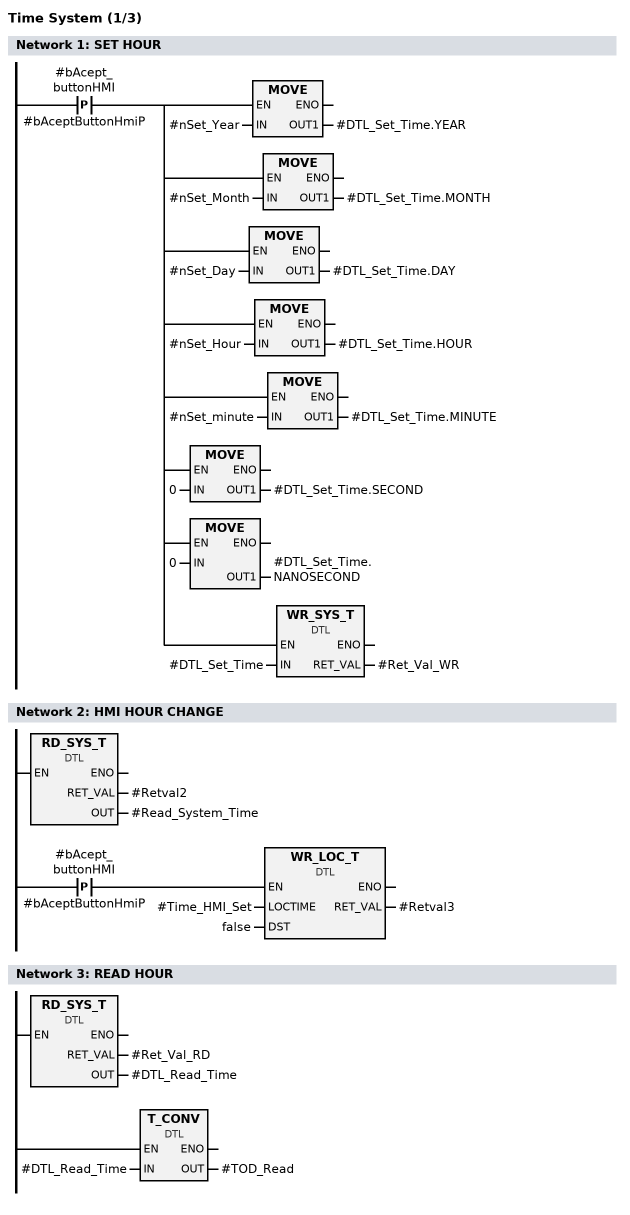
   RUNG wire#powerrail
      P_Contact(operand := #bAcept_buttonHMI, bit := #bAceptButtonHmiP)
      wire#w1
      Move(in := #nSet_Year, out1 => #DTL_Set_Time.YEAR)
   END_RUNG
   RUNG wire#w1
      Move(in := #nSet_Month, out1 => #DTL_Set_Time.MONTH)
   END_RUNG
   RUNG wire#w1
      Move(in := #nSet_Day, out1 => #DTL_Set_Time.DAY)
   END_RUNG
   RUNG wire#w1
      Move(in := #nSet_Hour, out1 => #DTL_Set_Time.HOUR)
   END_RUNG
   RUNG wire#w1
      Move(in := #nSet_minute, out1 => #DTL_Set_Time.MINUTE)
   END_RUNG
   RUNG wire#w1
      Move(in := 0, out1 => #DTL_Set_Time.SECOND)
   END_RUNG
   RUNG wire#w1
      Move(in := 0, out1 => #DTL_Set_Time.NANOSECOND)
   END_RUNG
   RUNG wire#w1
      { S7_Templates := "date_type := DTL" } WR_SYS_T(IN := #DTL_Set_Time, RET_VAL => #Ret_Val_WR)
   END_RUNG
   // the same network as SCL:
   #_w1 := #bAcept_buttonHMI AND NOT #bAceptButtonHmiP;   // rising edge of #bAcept_buttonHMI
   #bAceptButtonHmiP := #bAcept_buttonHMI;
   IF #_w1 THEN
       #DTL_Set_Time.YEAR := #nSet_Year;
       #DTL_Set_Time.MONTH := #nSet_Month;
       #DTL_Set_Time.DAY := #nSet_Day;
       #DTL_Set_Time.HOUR := #nSet_Hour;
       #DTL_Set_Time.MINUTE := #nSet_minute;
       #DTL_Set_Time.SECOND := 0;
       #DTL_Set_Time.NANOSECOND := 0;
       #Ret_Val_WR := WR_SYS_T(IN := #DTL_Set_Time);
   END_IF;
END_REGION

REGION Network 2: HMI HOUR CHANGE
   RUNG wire#powerrail
      { S7_Templates := "date_type := DTL" } RD_SYS_T(RET_VAL => #Retval2, OUT => #Read_System_Time)
   END_RUNG
   RUNG wire#powerrail
      P_Contact(operand := #bAcept_buttonHMI, bit := #bAceptButtonHmiP)
      { S7_Templates := "loctime_type := DTL" } WR_LOC_T(LOCTIME := #Time_HMI_Set, DST := false, Ret_Val => #Retval3)
   END_RUNG
   // the same network as SCL:
   #Retval2 := RD_SYS_T(OUT => #Read_System_Time);
   #_w1 := #bAcept_buttonHMI AND NOT #bAceptButtonHmiP;   // rising edge of #bAcept_buttonHMI
   #bAceptButtonHmiP := #bAcept_buttonHMI;
   IF #_w1 THEN #Retval3 := WR_LOC_T(LOCTIME := #Time_HMI_Set, DST := false); END_IF;
END_REGION

REGION Network 3: READ HOUR
   RUNG wire#powerrail
      { S7_Templates := "date_type := DTL" } RD_SYS_T(RET_VAL => #Ret_Val_RD, OUT => #DTL_Read_Time)
   END_RUNG
   RUNG wire#powerrail
      { S7_Templates := "[src_type := DTL, dest_type := Time_Of_Day]" } T_CONV(IN := #DTL_Read_Time, OUT => #TOD_Read)
   END_RUNG
   // the same network as SCL:
   #Ret_Val_RD := RD_SYS_T(OUT => #DTL_Read_Time);
   T_CONV(IN := #DTL_Read_Time, OUT => #TOD_Read);
END_REGION

REGION Network 4: WORK SHIFTS
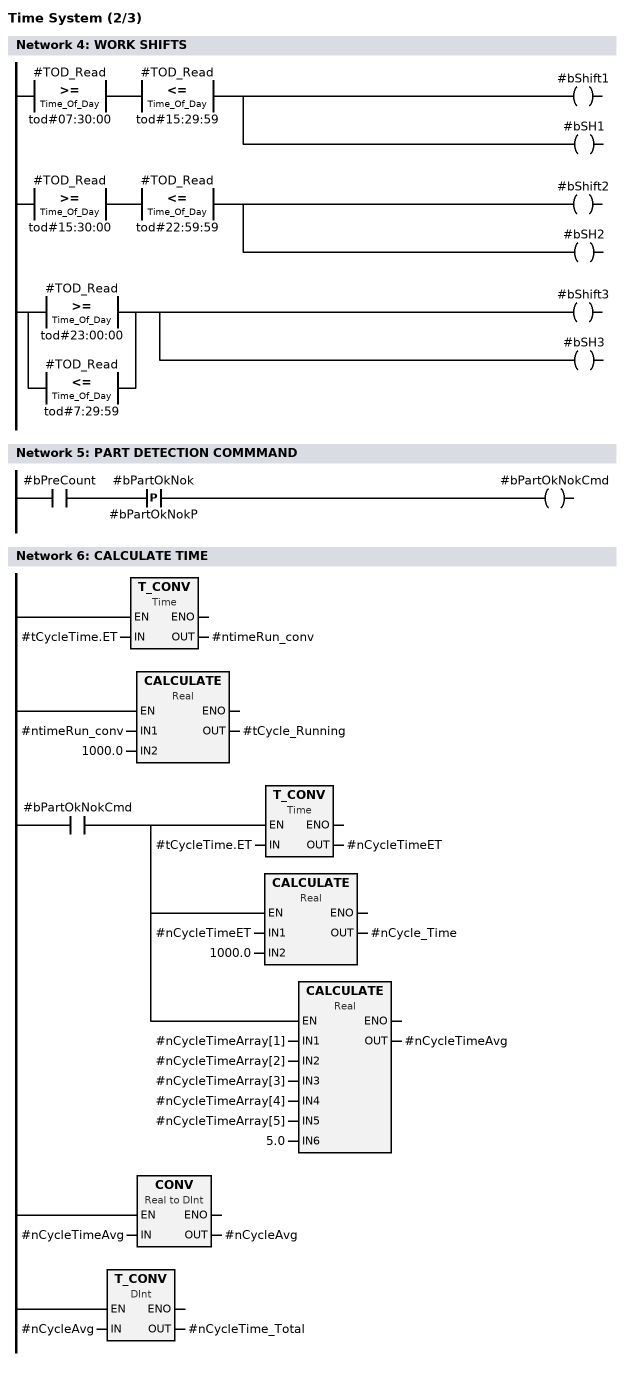
   RUNG wire#powerrail
      { S7_Templates := "SrcType := Time_Of_Day" } GE_Contact(in1 := #TOD_Read, in2 := tod#07:30:00)
      { S7_Templates := "SrcType := Time_Of_Day" } LE_Contact(in1 := #TOD_Read, in2 := tod#15:29:59)
      wire#w1
      Coil( #bShift1 )
   END_RUNG
   RUNG wire#w1
      Coil( #bSH1 )
   END_RUNG
   RUNG wire#powerrail
      { S7_Templates := "SrcType := Time_Of_Day" } GE_Contact(in1 := #TOD_Read, in2 := tod#15:30:00)
      { S7_Templates := "SrcType := Time_Of_Day" } LE_Contact(in1 := #TOD_Read, in2 := tod#22:59:59)
      wire#w2
      Coil( #bShift2 )
   END_RUNG
   RUNG wire#w2
      Coil( #bSH2 )
   END_RUNG
   RUNG wire#powerrail
      { S7_Templates := "SrcType := Time_Of_Day" } GE_Contact(in1 := #TOD_Read, in2 := tod#23:00:00)
      wire#w3
      Coil( #bShift3 )
   END_RUNG
   RUNG wire#powerrail
      { S7_Templates := "SrcType := Time_Of_Day" } LE_Contact(in1 := #TOD_Read, in2 := tod#7:29:59)
   END_RUNG wire#w3
   RUNG wire#w3
      Coil( #bSH3 )
   END_RUNG
   // the same network as SCL:
   #bShift1 := (#TOD_Read >= tod#07:30:00) AND (#TOD_Read <= tod#15:29:59);
   #bSH1 := #bShift1;
   #bShift2 := (#TOD_Read >= tod#15:30:00) AND (#TOD_Read <= tod#22:59:59);
   #bSH2 := #bShift2;
   #bShift3 := (#TOD_Read >= tod#23:00:00) OR (#TOD_Read <= tod#7:29:59);
   #bSH3 := #bShift3;
END_REGION

REGION Network 5: PART DETECTION COMMMAND
   RUNG wire#powerrail
      Contact( #bPreCount )
      P_Contact(operand := #bPartOkNok, bit := #bPartOkNokP)
      Coil( #bPartOkNokCmd )
   END_RUNG
   // the same network as SCL:
   #_w1 := #bPreCount AND #bPartOkNok AND NOT #bPartOkNokP;   // rising edge of #bPartOkNok
   #bPartOkNokP := #bPartOkNok;
   #bPartOkNokCmd := #_w1;
END_REGION

REGION Network 6: CALCULATE TIME
   RUNG wire#powerrail
      { S7_Templates := "[src_type := Time, dest_type := UDInt]" } T_CONV(IN := #tCycleTime.ET, OUT => #ntimeRun_conv)
   END_RUNG
   RUNG wire#powerrail
      { S7_Templates := "SrcType := Real"; S7_Expression := "in1/in2" } Calculate(in1 := #ntimeRun_conv, in2 := 1000.0, out => #tCycle_Running)
   END_RUNG
   RUNG wire#powerrail
      Contact( #bPartOkNokCmd )
      wire#w1
      { S7_Templates := "[src_type := Time, dest_type := UDInt]" } T_CONV(IN := #tCycleTime.ET, OUT => #nCycleTimeET)
   END_RUNG
   RUNG wire#w1
      { S7_Templates := "SrcType := Real"; S7_Expression := "in1/in2" } Calculate(in1 := #nCycleTimeET, in2 := 1000.0, out => #nCycle_Time)
   END_RUNG
   RUNG wire#w1
      { S7_Templates := "SrcType := Real"; S7_Expression := "(in1+in2+in3+in4+in5)/in6" } Calculate(in1 := #nCycleTimeArray[1], in2 := #nCycleTimeArray[2], in3 := #nCycleTimeArray[3], in4 := #nCycleTimeArray[4], in5 := #nCycleTimeArray[5], in6 := 5.0, out => #nCycleTimeAvg)
   END_RUNG
   RUNG wire#powerrail
      { S7_Templates := "[SrcType := Real, DestType := DInt]" } Convert(in := #nCycleTimeAvg, out => #nCycleAvg)
   END_RUNG
   RUNG wire#powerrail
      { S7_Templates := "[src_type := DInt, dest_type := Time_Of_Day]" } T_CONV(IN := #nCycleAvg, OUT => #nCycleTime_Total)
   END_RUNG
   // the same network as SCL:
   T_CONV(IN := #tCycleTime.ET, OUT => #ntimeRun_conv);
   #tCycle_Running := #ntimeRun_conv/1000.0;
   IF #bPartOkNokCmd THEN
       T_CONV(IN := #tCycleTime.ET, OUT => #nCycleTimeET);
       #nCycle_Time := #nCycleTimeET/1000.0;
       #nCycleTimeAvg := (#nCycleTimeArray[1]+#nCycleTimeArray[2]+#nCycleTimeArray[3]+#nCycleTimeArray[4]+#nCycleTimeArray[5])/5.0;
   END_IF;
   #nCycleAvg := REAL_TO_DINT(#nCycleTimeAvg);
   T_CONV(IN := #nCycleAvg, OUT => #nCycleTime_Total);
END_REGION

REGION Network 7: CICLE TIME ARRANGEMENT
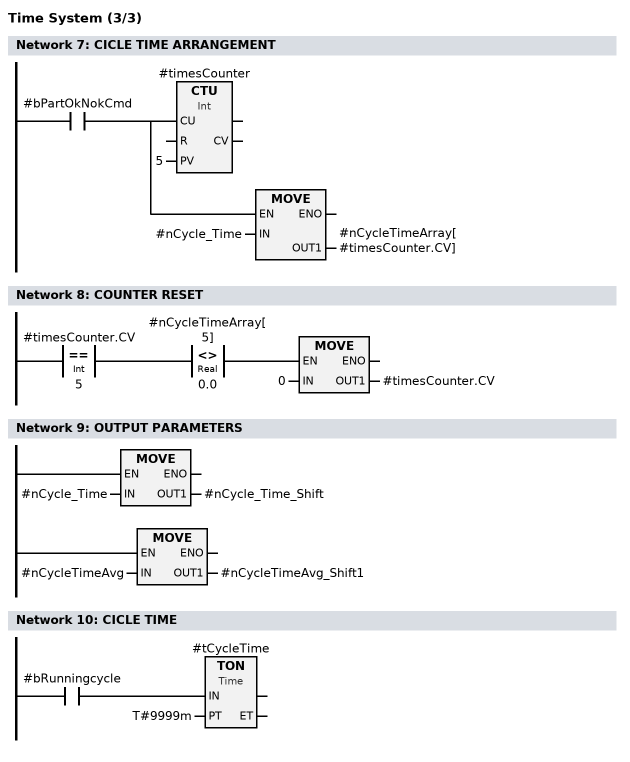
   RUNG wire#powerrail
      Contact( #bPartOkNokCmd )
      wire#w1
      { S7_Templates := "value_type := Int" } #timesCounter.CTU(r :=, pv := 5, cv =>)
   END_RUNG
   RUNG wire#w1
      Move(in := #nCycle_Time, out1 => #nCycleTimeArray[#timesCounter.CV])
   END_RUNG
   // the same network as SCL:
   #timesCounter.CTU(CU := #bPartOkNokCmd, PV := 5);
   IF #bPartOkNokCmd THEN #nCycleTimeArray[#timesCounter.CV] := #nCycle_Time; END_IF;
END_REGION

REGION Network 8: COUNTER RESET
   RUNG wire#powerrail
      { S7_Templates := "SrcType := Int" } EQ_Contact(in1 := #timesCounter.CV, in2 := 5)
      { S7_Templates := "SrcType := Real" } NE_Contact(in1 := #nCycleTimeArray[5], in2 := 0.0)
      Move(in := 0, out1 => #timesCounter.CV)
   END_RUNG
   // the same network as SCL:
   IF (#timesCounter.CV = 5) AND (#nCycleTimeArray[5] <> 0.0) THEN #timesCounter.CV := 0; END_IF;
END_REGION

REGION Network 9: OUTPUT PARAMETERS
   RUNG wire#powerrail
      Move(in := #nCycle_Time, out1 => #nCycle_Time_Shift)
   END_RUNG
   RUNG wire#powerrail
      Move(in := #nCycleTimeAvg, out1 => #nCycleTimeAvg_Shift1)
   END_RUNG
   // the same network as SCL:
   #nCycle_Time_Shift := #nCycle_Time;
   #nCycleTimeAvg_Shift1 := #nCycleTimeAvg;
END_REGION

REGION Network 10: CICLE TIME
   RUNG wire#powerrail
      Contact( #bRunningcycle )
      { S7_Templates := "time_type := Time" } #tCycleTime.TON(pt := T#9999m, et =>)
   END_RUNG
   // the same network as SCL:
   #tCycleTime.TON(IN := #bRunningcycle, PT := T#9999m);
END_REGION
END_FUNCTION_BLOCK

FUNCTION "FC_EKS" : Void   // FC305, LAD
TITLE = Euchner Management EKS KEY
{ S7_Optimized_Access := 'FALSE' }
VERSION : 0.1
// stored: AutoNumber false, IsIECCheckEnabled false, SetENOAutomatically false, UDAEnableTagReadback false
   VAR_INPUT
      iKEY_IN : Bool;
      iEKS_LEVEL : Byte;
      iEKS_EMPLOYEE_ID : DWord;
      iEKS_KEY_ID1 : DWord;
      iEKS_KEY_ID2 : DWord;
      iEKS_JOB_FINISHED : Bool;
      "Current_page_of HMI" : Word;
   END_VAR
   VAR_OUTPUT
      qEKS_START_ADDRESS : Byte;
      qEKS_DATA_LENGTH : Byte;
      qEKS_DATA_1 : Byte;
      qEKS_DATA_2 : DWord;
      qEKS_WRITE_CMD : Bool;
   END_VAR
   VAR_TEMP
      tNone : Bool;
      tDBAddressKeys : Int;
      tDBAddressHMIPage : Int;
      tDBKeyStructLength : Int;
      tDBAddress : Int;
      tDBLength : Int;
      tCycle : Int;
      tFill : Int;
      tKey : "udt_EKS_KEY";
      tDBStartAddress : Int;
      tsearch : Bool;
      i : Int;
   END_VAR
   VAR CONSTANT
      DB : Byte := 16#84;
   END_VAR
   VAR_TEMP   // added for the SCL form of the ladder/FBD networks
      _w1 : Bool;
      _w2 : Bool;
   END_VAR
BEGIN

REGION Network 1: Actual HMI page index limits
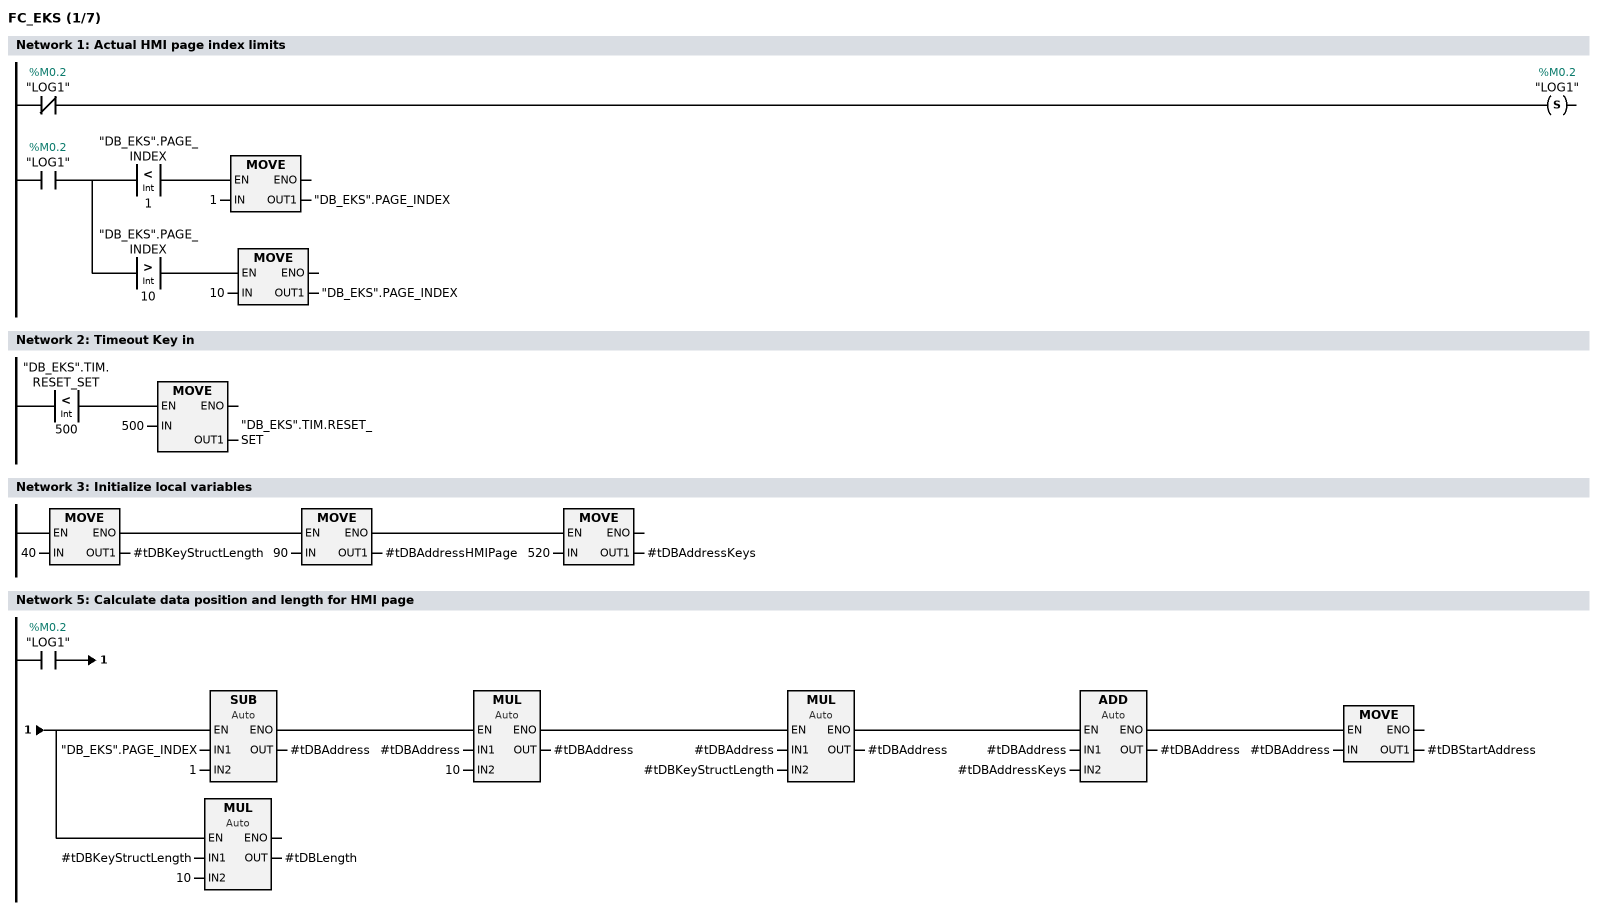
   RUNG wire#powerrail
      I_Contact( "LOG1" )
      S_Coil( "LOG1" )
   END_RUNG
   RUNG wire#powerrail
      Contact( "LOG1" )
      wire#w1
      { S7_Templates := "SrcType := Int" } LT_Contact(in1 := "DB_EKS".PAGE_INDEX, in2 := 1)
      Move(in := 1, out1 => "DB_EKS".PAGE_INDEX)
   END_RUNG
   RUNG wire#w1
      { S7_Templates := "SrcType := Int" } GT_Contact(in1 := "DB_EKS".PAGE_INDEX, in2 := 10)
      Move(in := 10, out1 => "DB_EKS".PAGE_INDEX)
   END_RUNG
   // the same network as SCL:
   IF NOT "LOG1" THEN "LOG1" := TRUE; END_IF;
   IF "LOG1" AND ("DB_EKS".PAGE_INDEX < 1) THEN "DB_EKS".PAGE_INDEX := 1; END_IF;
   IF "LOG1" AND ("DB_EKS".PAGE_INDEX > 10) THEN "DB_EKS".PAGE_INDEX := 10; END_IF;
END_REGION

REGION Network 2: Timeout Key in
   RUNG wire#powerrail
      { S7_Templates := "SrcType := Int" } LT_Contact(in1 := "DB_EKS".TIM.RESET_SET, in2 := 500)
      Move(in := 500, out1 => "DB_EKS".TIM.RESET_SET)
   END_RUNG
   // the same network as SCL:
   IF "DB_EKS".TIM.RESET_SET < 500 THEN "DB_EKS".TIM.RESET_SET := 500; END_IF;
END_REGION

REGION Network 3: Initialize local variables
   RUNG wire#powerrail
      Move(in := 40, out1 => #tDBKeyStructLength)
      Move(in := 90, out1 => #tDBAddressHMIPage)
      Move(in := 520, out1 => #tDBAddressKeys)
   END_RUNG
   // the same network as SCL:
   #tDBKeyStructLength := 40;
   #tDBAddressHMIPage := 90;
   #tDBAddressKeys := 520;
END_REGION

REGION Network 5: Calculate data position and length for HMI page
   RUNG wire#powerrail
      Contact( "LOG1" )
      wire#w1
      Sub(in1 := "DB_EKS".PAGE_INDEX, in2 := 1, out => #tDBAddress)
      Mul(in1 := #tDBAddress, in2 := 10, out => #tDBAddress)
      Mul(in1 := #tDBAddress, in2 := #tDBKeyStructLength, out => #tDBAddress)
      Add(in1 := #tDBAddress, in2 := #tDBAddressKeys, out => #tDBAddress)
      Move(in := #tDBAddress, out1 => #tDBStartAddress)
   END_RUNG
   RUNG wire#w1
      Mul(in1 := #tDBKeyStructLength, in2 := 10, out => #tDBLength)
   END_RUNG
   // the same network as SCL:
   IF "LOG1" THEN
       #tDBAddress := "DB_EKS".PAGE_INDEX - 1;
       #tDBAddress := #tDBAddress * 10;
       #tDBAddress := #tDBAddress * #tDBKeyStructLength;
       #tDBAddress := #tDBAddress + #tDBAddressKeys;
       #tDBStartAddress := #tDBAddress;
       #tDBLength := #tDBKeyStructLength * 10;
   END_IF;
END_REGION

REGION Network 6 (SCL): Copy data for page (10 keys)
   POKE_BLK(area_src:=#DB,
            dbNumber_src:=305,
            byteOffset_src:=#tDBAddress,
            area_dest:=#DB,
            dbNumber_dest:=305,
            byteOffset_dest:=90,
            count:=#tDBLength);
END_REGION

REGION Network 8: Inserted key
   // Store_Key_In is used to display only 1 time the level of euchner during storage function.
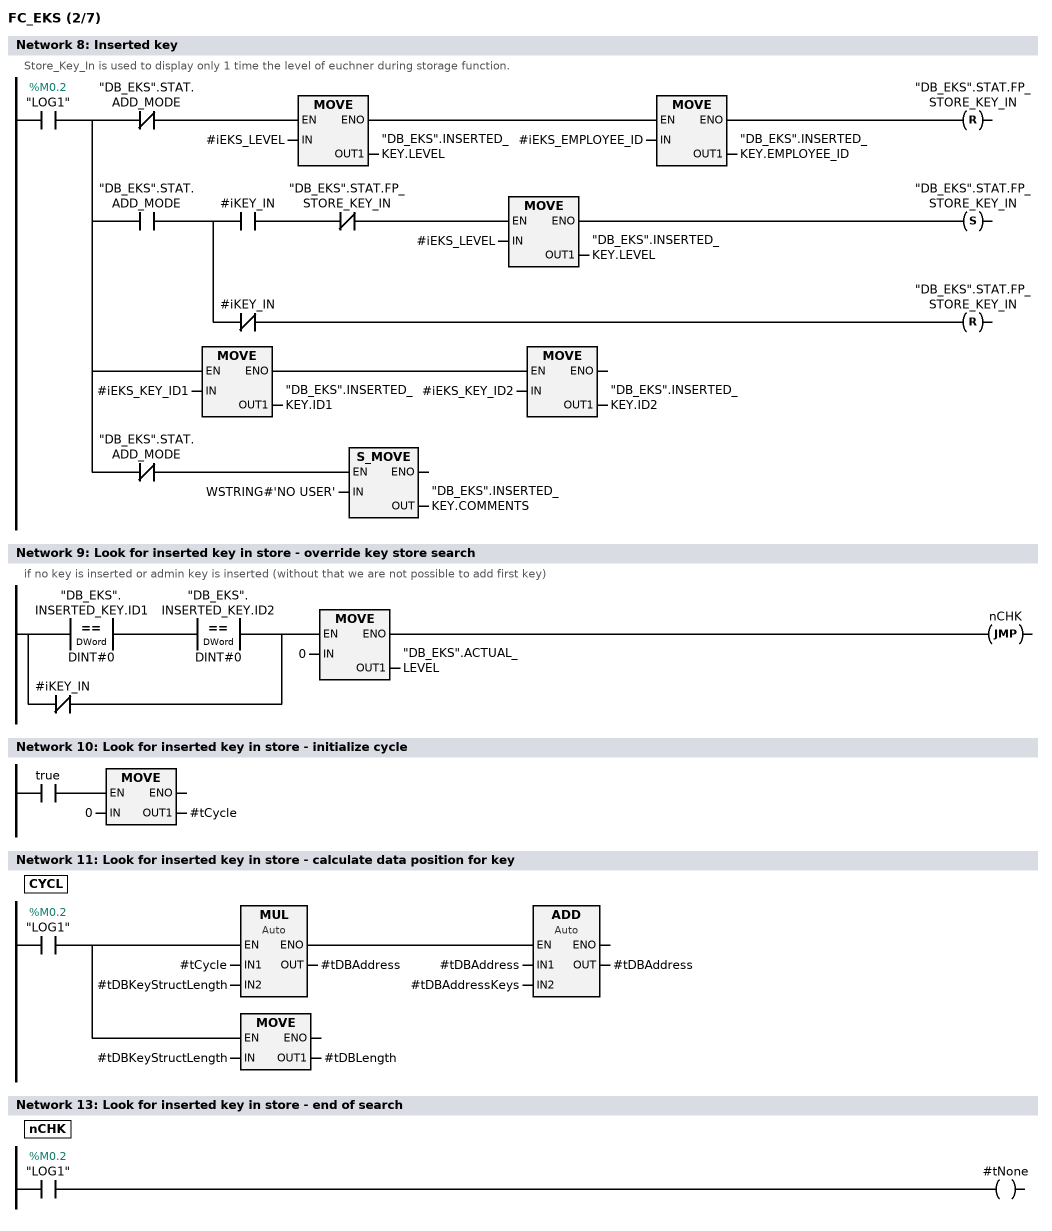
   RUNG wire#powerrail
      Contact( "LOG1" )
      wire#w1
      I_Contact( "DB_EKS".STAT.ADD_MODE )
      Move(in := #iEKS_LEVEL, out1 => "DB_EKS".INSERTED_KEY.LEVEL)
      Move(in := #iEKS_EMPLOYEE_ID, out1 => "DB_EKS".INSERTED_KEY.EMPLOYEE_ID)
      R_Coil( "DB_EKS".STAT.FP_STORE_KEY_IN )
   END_RUNG
   RUNG wire#w1
      Contact( "DB_EKS".STAT.ADD_MODE )
      wire#w2
      Contact( #iKEY_IN )
      I_Contact( "DB_EKS".STAT.FP_STORE_KEY_IN )
      Move(in := #iEKS_LEVEL, out1 => "DB_EKS".INSERTED_KEY.LEVEL)
      S_Coil( "DB_EKS".STAT.FP_STORE_KEY_IN )
   END_RUNG
   RUNG wire#w2
      I_Contact( #iKEY_IN )
      R_Coil( "DB_EKS".STAT.FP_STORE_KEY_IN )
   END_RUNG
   RUNG wire#w1
      Move(in := #iEKS_KEY_ID1, out1 => "DB_EKS".INSERTED_KEY.ID1)
      Move(in := #iEKS_KEY_ID2, out1 => "DB_EKS".INSERTED_KEY.ID2)
   END_RUNG
   RUNG wire#w1
      I_Contact( "DB_EKS".STAT.ADD_MODE )
      S_Move(in := WSTRING#'NO USER', out => "DB_EKS".INSERTED_KEY.COMMENTS)
   END_RUNG
   // the same network as SCL:
   IF "LOG1" AND NOT "DB_EKS".STAT.ADD_MODE THEN
       "DB_EKS".INSERTED_KEY.LEVEL := #iEKS_LEVEL;
       "DB_EKS".INSERTED_KEY.EMPLOYEE_ID := #iEKS_EMPLOYEE_ID;
       "DB_EKS".STAT.FP_STORE_KEY_IN := FALSE;
   END_IF;
   #_w1 := "LOG1" AND "DB_EKS".STAT.ADD_MODE;
   IF #_w1 AND #iKEY_IN AND NOT "DB_EKS".STAT.FP_STORE_KEY_IN THEN
       "DB_EKS".INSERTED_KEY.LEVEL := #iEKS_LEVEL;
       "DB_EKS".STAT.FP_STORE_KEY_IN := TRUE;
   END_IF;
   IF #_w1 AND NOT #iKEY_IN THEN "DB_EKS".STAT.FP_STORE_KEY_IN := FALSE; END_IF;
   IF "LOG1" THEN
       "DB_EKS".INSERTED_KEY.ID1 := #iEKS_KEY_ID1;
       "DB_EKS".INSERTED_KEY.ID2 := #iEKS_KEY_ID2;
   END_IF;
   IF "LOG1" AND NOT "DB_EKS".STAT.ADD_MODE THEN "DB_EKS".INSERTED_KEY.COMMENTS := WSTRING#'NO USER'; END_IF;
END_REGION

REGION Network 9: Look for inserted key in store - override key store search
   // if no key is inserted or admin key is inserted (without that we are not possible to add first key)
   RUNG wire#powerrail
      { S7_Templates := "SrcType := DWord" } EQ_Contact(in1 := "DB_EKS".INSERTED_KEY.ID1, in2 := DINT#0)
      { S7_Templates := "SrcType := DWord" } EQ_Contact(in1 := "DB_EKS".INSERTED_KEY.ID2, in2 := DINT#0)
      wire#w1
      Move(in := 0, out1 => "DB_EKS".ACTUAL_LEVEL)
      JumpCoil( nCHK )
   END_RUNG
   RUNG wire#powerrail
      I_Contact( #iKEY_IN )
   END_RUNG wire#w1
   // the same network as SCL:
   #_w1 := (("DB_EKS".INSERTED_KEY.ID1 = DINT#0) AND ("DB_EKS".INSERTED_KEY.ID2 = DINT#0)) OR NOT #iKEY_IN;
   IF #_w1 THEN
       "DB_EKS".ACTUAL_LEVEL := 0;
       GOTO nCHK;
   END_IF;
END_REGION

REGION Network 10: Look for inserted key in store - initialize cycle
   RUNG wire#powerrail
      Contact( true )
      Move(in := 0, out1 => #tCycle)
   END_RUNG
   // the same network as SCL:
   IF true THEN #tCycle := 0; END_IF;
END_REGION

REGION Network 11: Look for inserted key in store - calculate data position for key
   Label( CYCL )
   RUNG wire#powerrail
      Contact( "LOG1" )
      wire#w1
      Mul(in1 := #tCycle, in2 := #tDBKeyStructLength, out => #tDBAddress)
      Add(in1 := #tDBAddress, in2 := #tDBAddressKeys, out => #tDBAddress)
   END_RUNG
   RUNG wire#w1
      Move(in := #tDBKeyStructLength, out1 => #tDBLength)
   END_RUNG
   // the same network as SCL:
   CYCL:
   IF "LOG1" THEN
       #tDBAddress := #tCycle * #tDBKeyStructLength;
       #tDBAddress := #tDBAddress + #tDBAddressKeys;
       #tDBLength := #tDBKeyStructLength;
   END_IF;
END_REGION

REGION Network 12 (SCL): Look for inserted key in store - check ID of stored key
   FOR #i := 1 TO 130 DO
       #tKey := "DB_EKS".KEYS[#i];
       IF (#tKey.ID1 = "DB_EKS".INSERTED_KEY.ID1) AND
           (#tKey.ID2 = "DB_EKS".INSERTED_KEY.ID2) THEN
           "DB_EKS".ACTUAL_LEVEL := #tKey.LEVEL;
           "DB_EKS".INSERTED_KEY.COMMENTS := #tKey.COMMENTS;
           EXIT;
       END_IF;
   END_FOR;
END_REGION

REGION Network 13: Look for inserted key in store - end of search
   Label( nCHK )
   RUNG wire#powerrail
      Contact( "LOG1" )
      Coil( #tNone )
   END_RUNG
   // the same network as SCL:
   nCHK:
   #tNone := "LOG1";
END_REGION

REGION Network 14: Reset of EKS higher levels until key is removed
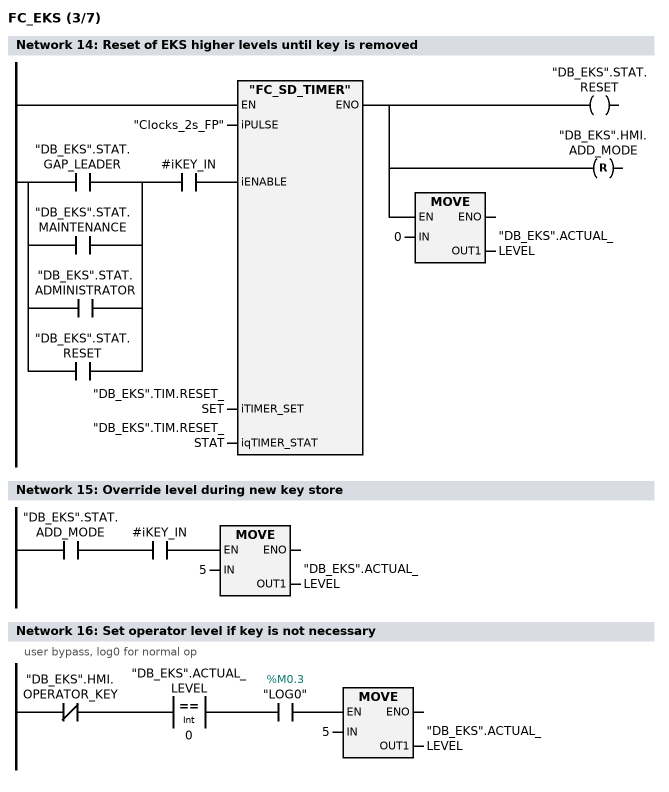
   RUNG wire#powerrail
      "FC_SD_TIMER"(iENABLE := wire#w2, iPULSE := "Clocks_2s_FP", iTIMER_SET := "DB_EKS".TIM.RESET_SET, iqTIMER_STAT := "DB_EKS".TIM.RESET_STAT)
      wire#w3
      Coil( "DB_EKS".STAT.RESET )
   END_RUNG
   RUNG wire#powerrail
      Contact( "DB_EKS".STAT.GAP_LEADER )
      wire#w1
      Contact( #iKEY_IN )
   END_RUNG wire#w2
   RUNG wire#powerrail
      Contact( "DB_EKS".STAT.MAINTENANCE )
   END_RUNG wire#w1
   RUNG wire#powerrail
      Contact( "DB_EKS".STAT.ADMINISTRATOR )
   END_RUNG wire#w1
   RUNG wire#powerrail
      Contact( "DB_EKS".STAT.RESET )
   END_RUNG wire#w1
   RUNG wire#w3
      R_Coil( "DB_EKS".HMI.ADD_MODE )
   END_RUNG
   RUNG wire#w3
      Move(in := 0, out1 => "DB_EKS".ACTUAL_LEVEL)
   END_RUNG
   // the same network as SCL:
   "FC_SD_TIMER"(iPULSE := "Clocks_2s_FP",
                 iENABLE := ("DB_EKS".STAT.GAP_LEADER OR "DB_EKS".STAT.MAINTENANCE OR "DB_EKS".STAT.ADMINISTRATOR OR "DB_EKS".STAT.RESET) AND #iKEY_IN,
                 iTIMER_SET := "DB_EKS".TIM.RESET_SET,
                 iqTIMER_STAT := "DB_EKS".TIM.RESET_STAT,
                 ENO => #_w1);
   "DB_EKS".STAT.RESET := #_w1;
   IF #_w1 THEN
       "DB_EKS".HMI.ADD_MODE := FALSE;
       "DB_EKS".ACTUAL_LEVEL := 0;
   END_IF;
END_REGION

REGION Network 15: Override level during new key store
   RUNG wire#powerrail
      Contact( "DB_EKS".STAT.ADD_MODE )
      Contact( #iKEY_IN )
      Move(in := 5, out1 => "DB_EKS".ACTUAL_LEVEL)
   END_RUNG
   // the same network as SCL:
   IF "DB_EKS".STAT.ADD_MODE AND #iKEY_IN THEN "DB_EKS".ACTUAL_LEVEL := 5; END_IF;
END_REGION

REGION Network 16: Set operator level if key is not necessary
   // user bypass, log0 for normal op
   RUNG wire#powerrail
      I_Contact( "DB_EKS".HMI.OPERATOR_KEY )
      { S7_Templates := "SrcType := Int" } EQ_Contact(in1 := "DB_EKS".ACTUAL_LEVEL, in2 := 0)
      Contact( "LOG0" )
      Move(in := 5, out1 => "DB_EKS".ACTUAL_LEVEL)
   END_RUNG
   // the same network as SCL:
   IF NOT "DB_EKS".HMI.OPERATOR_KEY AND ("DB_EKS".ACTUAL_LEVEL = 0) AND "LOG0" THEN
       "DB_EKS".ACTUAL_LEVEL := 5;
   END_IF;
END_REGION

REGION Network 17: EKS levels
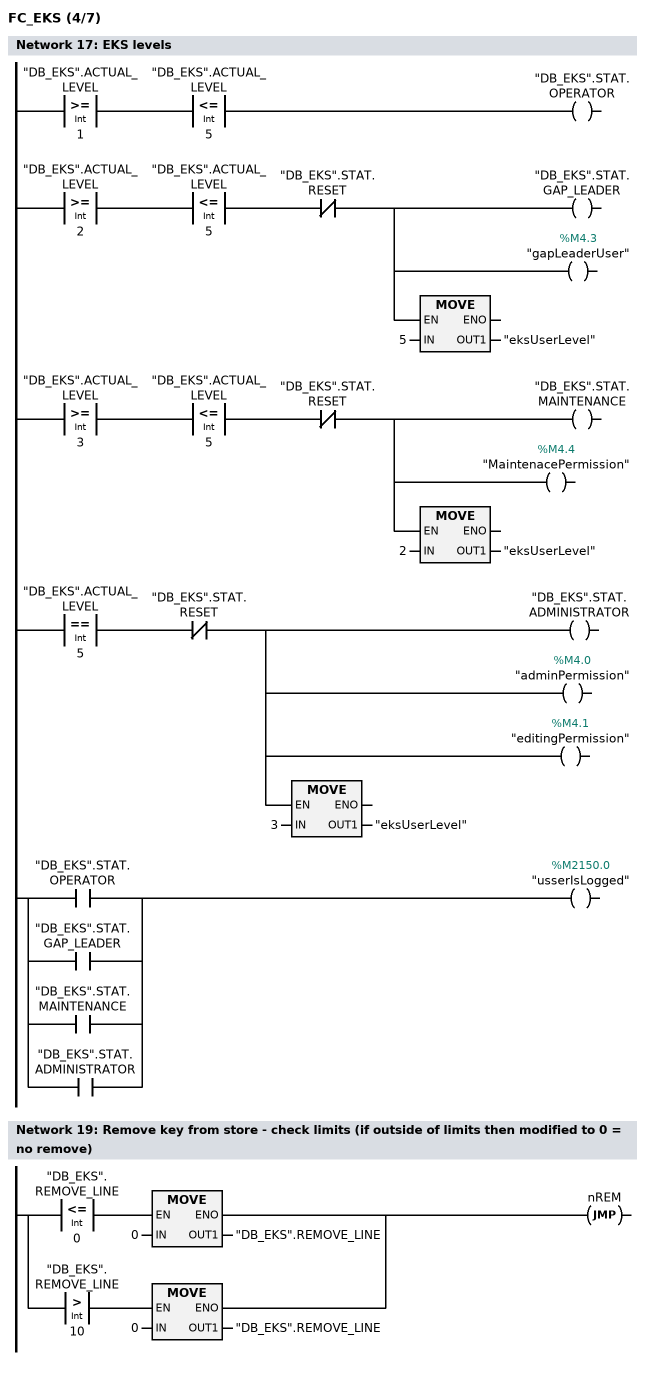
   RUNG wire#powerrail
      { S7_Templates := "SrcType := Int" } GE_Contact(in1 := "DB_EKS".ACTUAL_LEVEL, in2 := 1)
      { S7_Templates := "SrcType := Int" } LE_Contact(in1 := "DB_EKS".ACTUAL_LEVEL, in2 := 5)
      Coil( "DB_EKS".STAT.OPERATOR )
   END_RUNG
   RUNG wire#powerrail
      { S7_Templates := "SrcType := Int" } GE_Contact(in1 := "DB_EKS".ACTUAL_LEVEL, in2 := 2)
      { S7_Templates := "SrcType := Int" } LE_Contact(in1 := "DB_EKS".ACTUAL_LEVEL, in2 := 5)
      I_Contact( "DB_EKS".STAT.RESET )
      wire#w1
      Coil( "DB_EKS".STAT.GAP_LEADER )
   END_RUNG
   RUNG wire#w1
      Coil( "gapLeaderUser" )
   END_RUNG
   RUNG wire#w1
      Move(in := 5, out1 => "eksUserLevel")
   END_RUNG
   RUNG wire#powerrail
      { S7_Templates := "SrcType := Int" } GE_Contact(in1 := "DB_EKS".ACTUAL_LEVEL, in2 := 3)
      { S7_Templates := "SrcType := Int" } LE_Contact(in1 := "DB_EKS".ACTUAL_LEVEL, in2 := 5)
      I_Contact( "DB_EKS".STAT.RESET )
      wire#w2
      Coil( "DB_EKS".STAT.MAINTENANCE )
   END_RUNG
   RUNG wire#w2
      Coil( "MaintenacePermission" )
   END_RUNG
   RUNG wire#w2
      Move(in := 2, out1 => "eksUserLevel")
   END_RUNG
   RUNG wire#powerrail
      { S7_Templates := "SrcType := Int" } EQ_Contact(in1 := "DB_EKS".ACTUAL_LEVEL, in2 := 5)
      I_Contact( "DB_EKS".STAT.RESET )
      wire#w3
      Coil( "DB_EKS".STAT.ADMINISTRATOR )
   END_RUNG
   RUNG wire#w3
      Coil( "adminPermission" )
   END_RUNG
   RUNG wire#w3
      Coil( "editingPermission" )
   END_RUNG
   RUNG wire#w3
      Move(in := 3, out1 => "eksUserLevel")
   END_RUNG
   RUNG wire#powerrail
      Contact( "DB_EKS".STAT.OPERATOR )
      wire#w4
      Coil( "usserIsLogged" )
   END_RUNG
   RUNG wire#powerrail
      Contact( "DB_EKS".STAT.GAP_LEADER )
   END_RUNG wire#w4
   RUNG wire#powerrail
      Contact( "DB_EKS".STAT.MAINTENANCE )
   END_RUNG wire#w4
   RUNG wire#powerrail
      Contact( "DB_EKS".STAT.ADMINISTRATOR )
   END_RUNG wire#w4
   // the same network as SCL:
   "DB_EKS".STAT.OPERATOR := ("DB_EKS".ACTUAL_LEVEL >= 1) AND ("DB_EKS".ACTUAL_LEVEL <= 5);
   "DB_EKS".STAT.GAP_LEADER := ("DB_EKS".ACTUAL_LEVEL >= 2) AND ("DB_EKS".ACTUAL_LEVEL <= 5) AND NOT "DB_EKS".STAT.RESET;
   "gapLeaderUser" := "DB_EKS".STAT.GAP_LEADER;
   IF "DB_EKS".STAT.GAP_LEADER THEN "eksUserLevel" := 5; END_IF;
   "DB_EKS".STAT.MAINTENANCE := ("DB_EKS".ACTUAL_LEVEL >= 3) AND ("DB_EKS".ACTUAL_LEVEL <= 5) AND NOT "DB_EKS".STAT.RESET;
   "MaintenacePermission" := "DB_EKS".STAT.MAINTENANCE;
   IF "DB_EKS".STAT.MAINTENANCE THEN "eksUserLevel" := 2; END_IF;
   "DB_EKS".STAT.ADMINISTRATOR := ("DB_EKS".ACTUAL_LEVEL = 5) AND NOT "DB_EKS".STAT.RESET;
   "adminPermission" := "DB_EKS".STAT.ADMINISTRATOR;
   "editingPermission" := "DB_EKS".STAT.ADMINISTRATOR;
   IF "DB_EKS".STAT.ADMINISTRATOR THEN "eksUserLevel" := 3; END_IF;
   "usserIsLogged" := "DB_EKS".STAT.OPERATOR OR "DB_EKS".STAT.GAP_LEADER OR "DB_EKS".STAT.MAINTENANCE OR "DB_EKS".STAT.ADMINISTRATOR;
END_REGION

REGION Network 19: Remove key from store - check limits (if outside of limits then modified to 0 = no remove)
   RUNG wire#powerrail
      { S7_Templates := "SrcType := Int" } LE_Contact(in1 := "DB_EKS".REMOVE_LINE, in2 := 0)
      Move(in := 0, out1 => "DB_EKS".REMOVE_LINE)
      wire#w1
      JumpCoil( nREM )
   END_RUNG
   RUNG wire#powerrail
      { S7_Templates := "SrcType := Int" } GT_Contact(in1 := "DB_EKS".REMOVE_LINE, in2 := 10)
      Move(in := 0, out1 => "DB_EKS".REMOVE_LINE)
   END_RUNG wire#w1
   // the same network as SCL:
   #_w1 := "DB_EKS".REMOVE_LINE <= 0;
   IF #_w1 THEN "DB_EKS".REMOVE_LINE := 0; END_IF;
   #_w2 := "DB_EKS".REMOVE_LINE > 10;
   IF #_w2 THEN "DB_EKS".REMOVE_LINE := 0; END_IF;
   IF #_w1 OR #_w2 THEN GOTO nREM; END_IF;
END_REGION

REGION Network 20: Remove key from store - calculate data position and length for HMI page
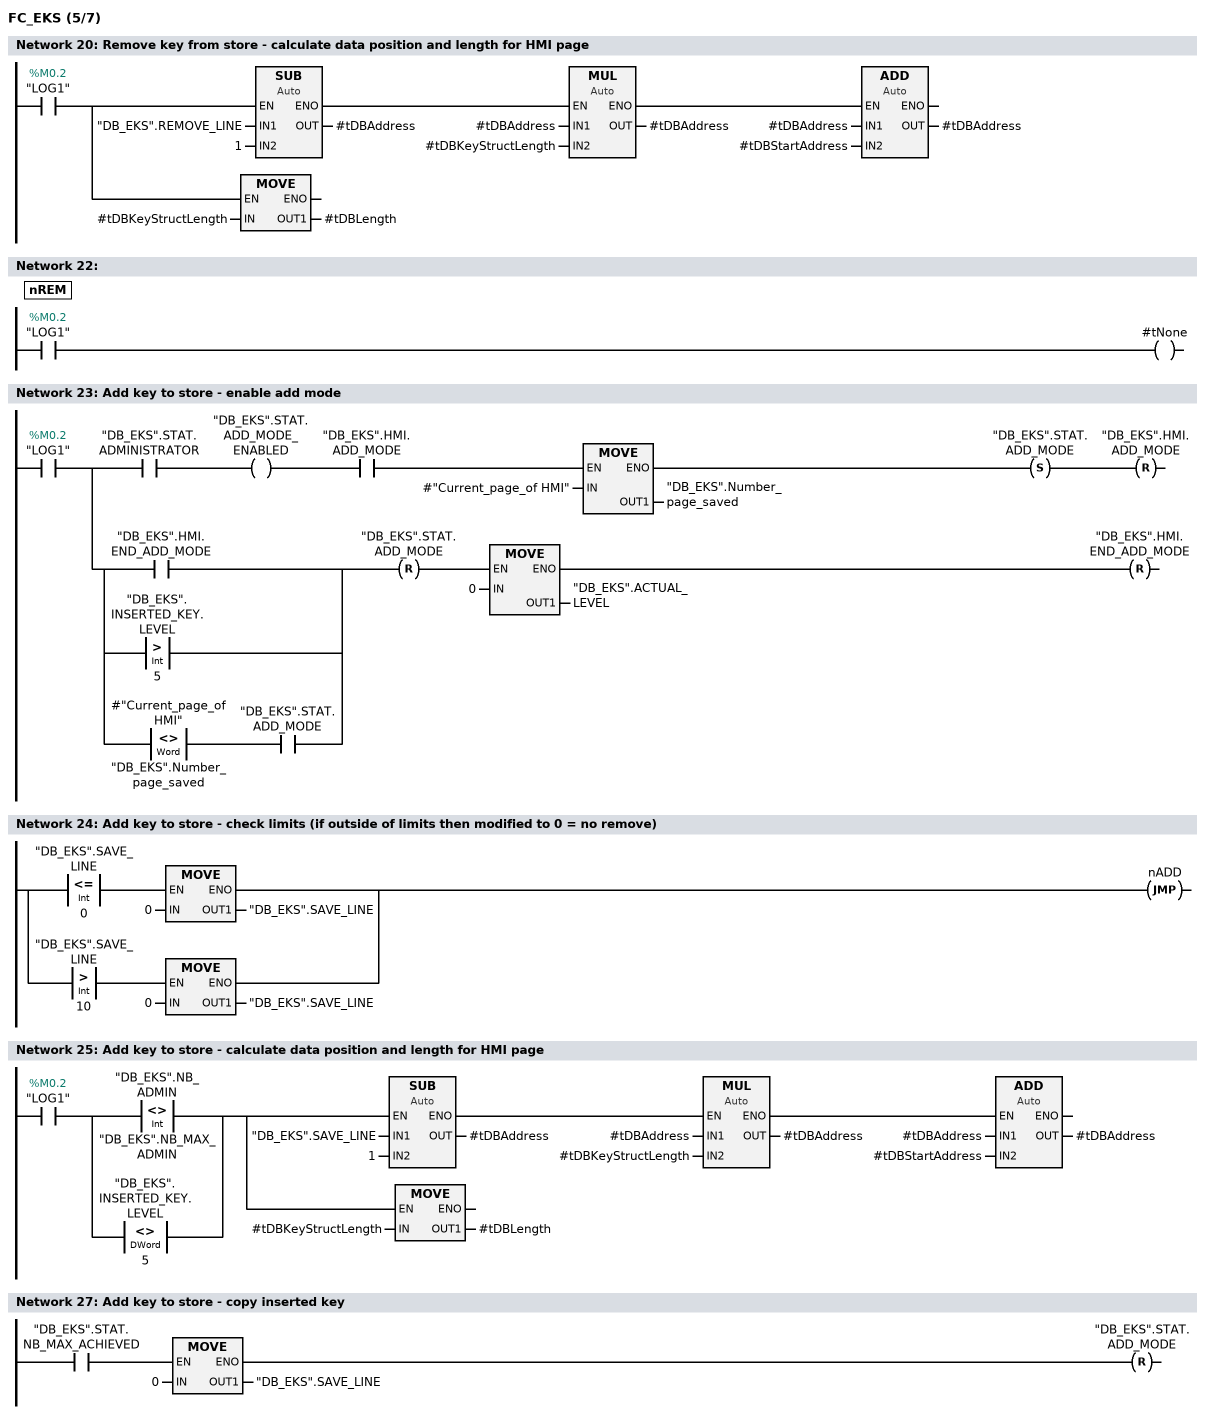
   RUNG wire#powerrail
      Contact( "LOG1" )
      wire#w1
      Sub(in1 := "DB_EKS".REMOVE_LINE, in2 := 1, out => #tDBAddress)
      Mul(in1 := #tDBAddress, in2 := #tDBKeyStructLength, out => #tDBAddress)
      Add(in1 := #tDBAddress, in2 := #tDBStartAddress, out => #tDBAddress)
   END_RUNG
   RUNG wire#w1
      Move(in := #tDBKeyStructLength, out1 => #tDBLength)
   END_RUNG
   // the same network as SCL:
   IF "LOG1" THEN
       #tDBAddress := "DB_EKS".REMOVE_LINE - 1;
       #tDBAddress := #tDBAddress * #tDBKeyStructLength;
       #tDBAddress := #tDBAddress + #tDBStartAddress;
       #tDBLength := #tDBKeyStructLength;
   END_IF;
END_REGION

REGION Network 21 (SCL): Remove key from store - delete key
   #tFill := 0;

   POKE_BLK(area_src:=#DB,
            dbNumber_src:=305,
            byteOffset_src:=5720,
            area_dest:=#DB,
            dbNumber_dest:=305,
            byteOffset_dest:=#tDBAddress,
            count:=#tDBLength);

   "DB_EKS".REMOVE_LINE := 0;
END_REGION

REGION Network 22
   Label( nREM )
   RUNG wire#powerrail
      Contact( "LOG1" )
      Coil( #tNone )
   END_RUNG
   // the same network as SCL:
   nREM:
   #tNone := "LOG1";
END_REGION

REGION Network 23: Add key to store - enable add mode
   RUNG wire#powerrail
      Contact( "LOG1" )
      wire#w1
      Contact( "DB_EKS".STAT.ADMINISTRATOR )
      Coil( "DB_EKS".STAT.ADD_MODE_ENABLED )
      Contact( "DB_EKS".HMI.ADD_MODE )
      Move(in := #"Current_page_of HMI", out1 => "DB_EKS".Number_page_saved)
      S_Coil( "DB_EKS".STAT.ADD_MODE )
      R_Coil( "DB_EKS".HMI.ADD_MODE )
   END_RUNG
   RUNG wire#w1
      Contact( "DB_EKS".HMI.END_ADD_MODE )
      wire#w2
      R_Coil( "DB_EKS".STAT.ADD_MODE )
      Move(in := 0, out1 => "DB_EKS".ACTUAL_LEVEL)
      R_Coil( "DB_EKS".HMI.END_ADD_MODE )
   END_RUNG
   RUNG wire#w1
      { S7_Templates := "SrcType := Int" } GT_Contact(in1 := "DB_EKS".INSERTED_KEY.LEVEL, in2 := 5)
   END_RUNG wire#w2
   RUNG wire#w1
      { S7_Templates := "SrcType := Word" } NE_Contact(in1 := #"Current_page_of HMI", in2 := "DB_EKS".Number_page_saved)
      Contact( "DB_EKS".STAT.ADD_MODE )
   END_RUNG wire#w2
   // the same network as SCL:
   "DB_EKS".STAT.ADD_MODE_ENABLED := "LOG1" AND "DB_EKS".STAT.ADMINISTRATOR;
   IF "DB_EKS".STAT.ADD_MODE_ENABLED AND "DB_EKS".HMI.ADD_MODE THEN
       "DB_EKS".Number_page_saved := #"Current_page_of HMI";
       "DB_EKS".STAT.ADD_MODE := TRUE;
       "DB_EKS".HMI.ADD_MODE := FALSE;
   END_IF;
   #_w1 := "LOG1" AND ("DB_EKS".HMI.END_ADD_MODE OR ("DB_EKS".INSERTED_KEY.LEVEL > 5) OR ((#"Current_page_of HMI" <> "DB_EKS".Number_page_saved) AND "DB_EKS".STAT.ADD_MODE));
   IF #_w1 THEN
       "DB_EKS".STAT.ADD_MODE := FALSE;
       "DB_EKS".ACTUAL_LEVEL := 0;
       "DB_EKS".HMI.END_ADD_MODE := FALSE;
   END_IF;
END_REGION

REGION Network 24: Add key to store - check limits (if outside of limits then modified to 0 = no remove)
   RUNG wire#powerrail
      { S7_Templates := "SrcType := Int" } LE_Contact(in1 := "DB_EKS".SAVE_LINE, in2 := 0)
      Move(in := 0, out1 => "DB_EKS".SAVE_LINE)
      wire#w1
      JumpCoil( nADD )
   END_RUNG
   RUNG wire#powerrail
      { S7_Templates := "SrcType := Int" } GT_Contact(in1 := "DB_EKS".SAVE_LINE, in2 := 10)
      Move(in := 0, out1 => "DB_EKS".SAVE_LINE)
   END_RUNG wire#w1
   // the same network as SCL:
   #_w1 := "DB_EKS".SAVE_LINE <= 0;
   IF #_w1 THEN "DB_EKS".SAVE_LINE := 0; END_IF;
   #_w2 := "DB_EKS".SAVE_LINE > 10;
   IF #_w2 THEN "DB_EKS".SAVE_LINE := 0; END_IF;
   IF #_w1 OR #_w2 THEN GOTO nADD; END_IF;
END_REGION

REGION Network 25: Add key to store - calculate data position and length for HMI page
   RUNG wire#powerrail
      Contact( "LOG1" )
      wire#w1
      { S7_Templates := "SrcType := Int" } NE_Contact(in1 := "DB_EKS".NB_ADMIN, in2 := "DB_EKS".NB_MAX_ADMIN)
      wire#w2
      Sub(in1 := "DB_EKS".SAVE_LINE, in2 := 1, out => #tDBAddress)
      Mul(in1 := #tDBAddress, in2 := #tDBKeyStructLength, out => #tDBAddress)
      Add(in1 := #tDBAddress, in2 := #tDBStartAddress, out => #tDBAddress)
   END_RUNG
   RUNG wire#w1
      { S7_Templates := "SrcType := DWord" } NE_Contact(in1 := "DB_EKS".INSERTED_KEY.LEVEL, in2 := 5)
   END_RUNG wire#w2
   RUNG wire#w2
      Move(in := #tDBKeyStructLength, out1 => #tDBLength)
   END_RUNG
   // the same network as SCL:
   IF "LOG1" AND (("DB_EKS".NB_ADMIN <> "DB_EKS".NB_MAX_ADMIN) OR ("DB_EKS".INSERTED_KEY.LEVEL <> 5)) THEN
       #tDBAddress := "DB_EKS".SAVE_LINE - 1;
       #tDBAddress := #tDBAddress * #tDBKeyStructLength;
       #tDBAddress := #tDBAddress + #tDBStartAddress;
       #tDBLength := #tDBKeyStructLength;
   END_IF;
END_REGION

REGION Network 26 (SCL): Add key to store - copy inserted key
   IF ("DB_EKS".INSERTED_KEY.LEVEL = 5  & NOT "DB_EKS".STAT.NB_MAX_ACHIEVED) OR
       ("DB_EKS".INSERTED_KEY.LEVEL <> 5) THEN
       POKE_BLK(area_src := #DB,
                dbNumber_src := 305,
                byteOffset_src := 50,
                area_dest := #DB,
                dbNumber_dest := 305,
                byteOffset_dest := #tDBAddress,
                count := #tDBLength);
      "DB_EKS".SAVE_LINE := 0;
   END_IF;
END_REGION

REGION Network 27: Add key to store - copy inserted key
   RUNG wire#powerrail
      Contact( "DB_EKS".STAT.NB_MAX_ACHIEVED )
      Move(in := 0, out1 => "DB_EKS".SAVE_LINE)
      R_Coil( "DB_EKS".STAT.ADD_MODE )
   END_RUNG
   // the same network as SCL:
   IF "DB_EKS".STAT.NB_MAX_ACHIEVED THEN
       "DB_EKS".SAVE_LINE := 0;
       "DB_EKS".STAT.ADD_MODE := FALSE;
   END_IF;
END_REGION

REGION Network 28
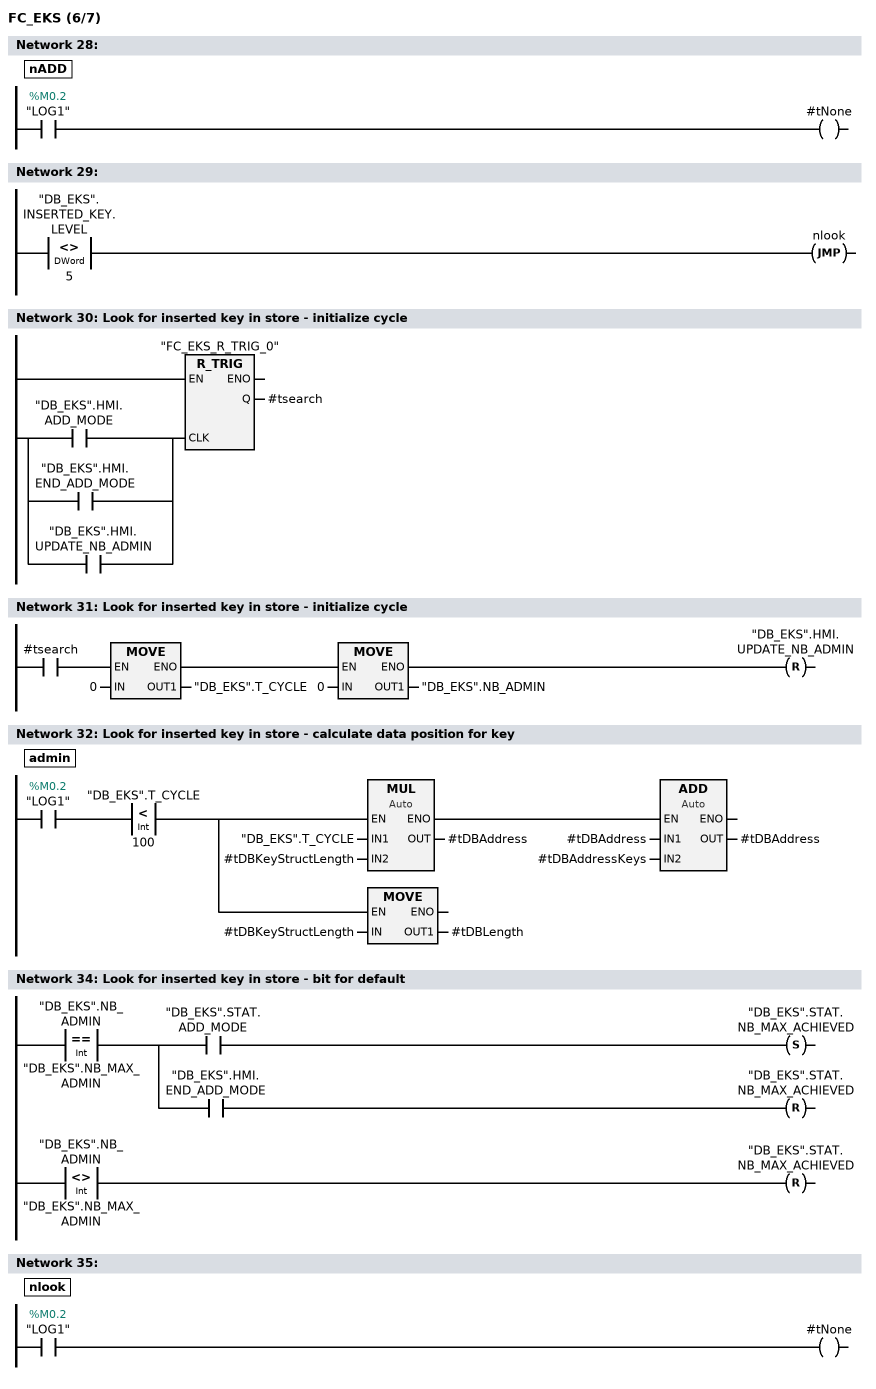
   Label( nADD )
   RUNG wire#powerrail
      Contact( "LOG1" )
      Coil( #tNone )
   END_RUNG
   // the same network as SCL:
   nADD:
   #tNone := "LOG1";
END_REGION

REGION Network 29
   RUNG wire#powerrail
      { S7_Templates := "SrcType := DWord" } NE_Contact(in1 := "DB_EKS".INSERTED_KEY.LEVEL, in2 := 5)
      JumpCoil( nlook )
   END_RUNG
   // the same network as SCL:
   IF "DB_EKS".INSERTED_KEY.LEVEL <> 5 THEN GOTO nlook; END_IF;
END_REGION

REGION Network 30: Look for inserted key in store - initialize cycle
   RUNG wire#powerrail
      "FC_EKS_R_TRIG_0".R_TRIG(CLK := wire#w1, Q => #tsearch)
   END_RUNG
   RUNG wire#powerrail
      Contact( "DB_EKS".HMI.ADD_MODE )
   END_RUNG wire#w1
   RUNG wire#powerrail
      Contact( "DB_EKS".HMI.END_ADD_MODE )
   END_RUNG wire#w1
   RUNG wire#powerrail
      Contact( "DB_EKS".HMI.UPDATE_NB_ADMIN )
   END_RUNG wire#w1
   // the same network as SCL:
   "FC_EKS_R_TRIG_0"(CLK := "DB_EKS".HMI.ADD_MODE OR "DB_EKS".HMI.END_ADD_MODE OR "DB_EKS".HMI.UPDATE_NB_ADMIN,   // R_TRIG
                     Q => #tsearch);
END_REGION

REGION Network 31: Look for inserted key in store - initialize cycle
   RUNG wire#powerrail
      Contact( #tsearch )
      Move(in := 0, out1 => "DB_EKS".T_CYCLE)
      Move(in := 0, out1 => "DB_EKS".NB_ADMIN)
      R_Coil( "DB_EKS".HMI.UPDATE_NB_ADMIN )
   END_RUNG
   // the same network as SCL:
   IF #tsearch THEN
       "DB_EKS".T_CYCLE := 0;
       "DB_EKS".NB_ADMIN := 0;
       "DB_EKS".HMI.UPDATE_NB_ADMIN := FALSE;
   END_IF;
END_REGION

REGION Network 32: Look for inserted key in store - calculate data position for key
   Label( admin )
   RUNG wire#powerrail
      Contact( "LOG1" )
      { S7_Templates := "SrcType := Int" } LT_Contact(in1 := "DB_EKS".T_CYCLE, in2 := 100)
      wire#w1
      Mul(in1 := "DB_EKS".T_CYCLE, in2 := #tDBKeyStructLength, out => #tDBAddress)
      Add(in1 := #tDBAddress, in2 := #tDBAddressKeys, out => #tDBAddress)
   END_RUNG
   RUNG wire#w1
      Move(in := #tDBKeyStructLength, out1 => #tDBLength)
   END_RUNG
   // the same network as SCL:
   admin:
   IF "LOG1" AND ("DB_EKS".T_CYCLE < 100) THEN
       #tDBAddress := "DB_EKS".T_CYCLE * #tDBKeyStructLength;
       #tDBAddress := #tDBAddress + #tDBAddressKeys;
       #tDBLength := #tDBKeyStructLength;
   END_IF;
END_REGION

REGION Network 33 (SCL): Look for inserted key in store - check ID of stored key
   FOR #i := 1 TO 100 DO
       #tKey := "DB_EKS".KEYS[#i];
       IF #tKey.LEVEL = 5 THEN
           "DB_EKS".NB_ADMIN += 1;
           CONTINUE;
       END_IF;
   END_FOR;
END_REGION

REGION Network 34: Look for inserted key in store - bit for default
   RUNG wire#powerrail
      { S7_Templates := "SrcType := Int" } EQ_Contact(in1 := "DB_EKS".NB_ADMIN, in2 := "DB_EKS".NB_MAX_ADMIN)
      wire#w1
      Contact( "DB_EKS".STAT.ADD_MODE )
      S_Coil( "DB_EKS".STAT.NB_MAX_ACHIEVED )
   END_RUNG
   RUNG wire#w1
      Contact( "DB_EKS".HMI.END_ADD_MODE )
      R_Coil( "DB_EKS".STAT.NB_MAX_ACHIEVED )
   END_RUNG
   RUNG wire#powerrail
      { S7_Templates := "SrcType := Int" } NE_Contact(in1 := "DB_EKS".NB_ADMIN, in2 := "DB_EKS".NB_MAX_ADMIN)
      R_Coil( "DB_EKS".STAT.NB_MAX_ACHIEVED )
   END_RUNG
   // the same network as SCL:
   #_w1 := "DB_EKS".NB_ADMIN = "DB_EKS".NB_MAX_ADMIN;
   IF #_w1 AND "DB_EKS".STAT.ADD_MODE THEN "DB_EKS".STAT.NB_MAX_ACHIEVED := TRUE; END_IF;
   IF #_w1 AND "DB_EKS".HMI.END_ADD_MODE THEN "DB_EKS".STAT.NB_MAX_ACHIEVED := FALSE; END_IF;
   IF "DB_EKS".NB_ADMIN <> "DB_EKS".NB_MAX_ADMIN THEN "DB_EKS".STAT.NB_MAX_ACHIEVED := FALSE; END_IF;
END_REGION

REGION Network 35
   Label( nlook )
   RUNG wire#powerrail
      Contact( "LOG1" )
      Coil( #tNone )
   END_RUNG
   // the same network as SCL:
   nlook:
   #tNone := "LOG1";
END_REGION

REGION Network 36: Write Level and Employer ID on Key
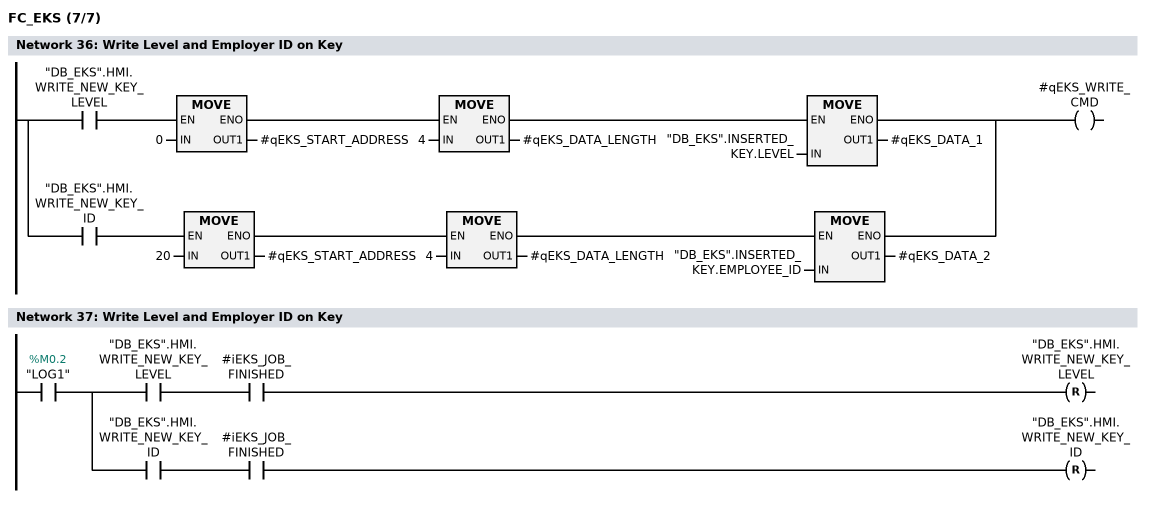
   RUNG wire#powerrail
      Contact( "DB_EKS".HMI.WRITE_NEW_KEY_LEVEL )
      Move(in := 0, out1 => #qEKS_START_ADDRESS)
      Move(in := 4, out1 => #qEKS_DATA_LENGTH)
      Move(in := "DB_EKS".INSERTED_KEY.LEVEL, out1 => #qEKS_DATA_1)
      wire#w1
      Coil( #qEKS_WRITE_CMD )
   END_RUNG
   RUNG wire#powerrail
      Contact( "DB_EKS".HMI.WRITE_NEW_KEY_ID )
      Move(in := 20, out1 => #qEKS_START_ADDRESS)
      Move(in := 4, out1 => #qEKS_DATA_LENGTH)
      Move(in := "DB_EKS".INSERTED_KEY.EMPLOYEE_ID, out1 => #qEKS_DATA_2)
   END_RUNG wire#w1
   // the same network as SCL:
   IF "DB_EKS".HMI.WRITE_NEW_KEY_LEVEL THEN
       #qEKS_START_ADDRESS := 0;
       #qEKS_DATA_LENGTH := 4;
       #qEKS_DATA_1 := "DB_EKS".INSERTED_KEY.LEVEL;
   END_IF;
   IF "DB_EKS".HMI.WRITE_NEW_KEY_ID THEN
       #qEKS_START_ADDRESS := 20;
       #qEKS_DATA_LENGTH := 4;
       #qEKS_DATA_2 := "DB_EKS".INSERTED_KEY.EMPLOYEE_ID;
   END_IF;
   #qEKS_WRITE_CMD := "DB_EKS".HMI.WRITE_NEW_KEY_LEVEL OR "DB_EKS".HMI.WRITE_NEW_KEY_ID;
END_REGION

REGION Network 37: Write Level and Employer ID on Key
   RUNG wire#powerrail
      Contact( "LOG1" )
      wire#w1
      Contact( "DB_EKS".HMI.WRITE_NEW_KEY_LEVEL )
      Contact( #iEKS_JOB_FINISHED )
      R_Coil( "DB_EKS".HMI.WRITE_NEW_KEY_LEVEL )
   END_RUNG
   RUNG wire#w1
      Contact( "DB_EKS".HMI.WRITE_NEW_KEY_ID )
      Contact( #iEKS_JOB_FINISHED )
      R_Coil( "DB_EKS".HMI.WRITE_NEW_KEY_ID )
   END_RUNG
   // the same network as SCL:
   IF "LOG1" AND "DB_EKS".HMI.WRITE_NEW_KEY_LEVEL AND #iEKS_JOB_FINISHED THEN
       "DB_EKS".HMI.WRITE_NEW_KEY_LEVEL := FALSE;
   END_IF;
   IF "LOG1" AND "DB_EKS".HMI.WRITE_NEW_KEY_ID AND #iEKS_JOB_FINISHED THEN
       "DB_EKS".HMI.WRITE_NEW_KEY_ID := FALSE;
   END_IF;
END_REGION
END_FUNCTION

FUNCTION "FC_SD_TIMER" : Void   // FC401, LAD
TITLE = Standard simple SD timer
{ S7_Optimized_Access := 'FALSE' }
FAMILY : system
VERSION : 1.0
// stored: AutoNumber false, IsIECCheckEnabled false, SetENOAutomatically false, UDAEnableTagReadback false
   VAR_INPUT
      iPULSE : Bool;   // time impulse
      iENABLE : Bool;   // release of timer
      iTIMER_SET : Int;   // preset value
   END_VAR
   VAR_IN_OUT
      iqTIMER_STAT : Int;   // actual value
   END_VAR
   VAR_TEMP
      tOk : Bool;
   END_VAR
BEGIN

REGION Network 1: If not enabled, then reset actual value of timer
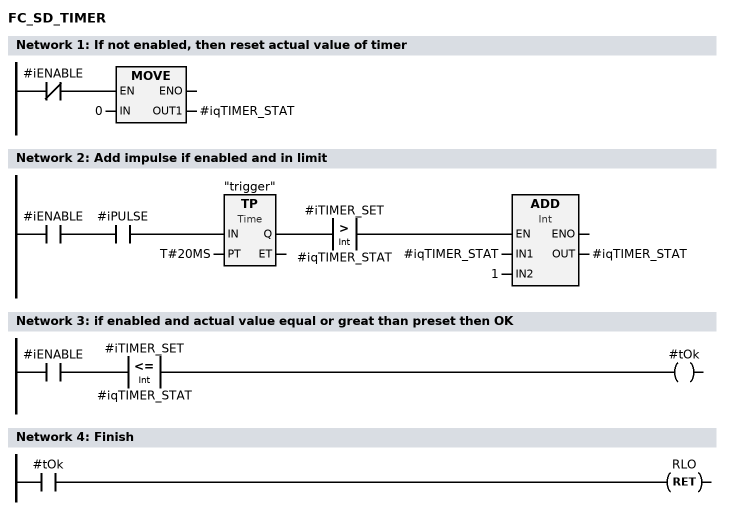
   RUNG wire#powerrail
      I_Contact( #iENABLE )
      { S7_GenerateENO := "TRUE" } Move(in := 0, out1 => #iqTIMER_STAT)
   END_RUNG
   // the same network as SCL:
   IF NOT #iENABLE THEN #iqTIMER_STAT := 0; END_IF;
END_REGION

REGION Network 2: Add impulse if enabled and in limit
   RUNG wire#powerrail
      Contact( #iENABLE )
      Contact( #iPULSE )
      { S7_Templates := "time_type := Time" } "trigger".TP(pt := T#20MS, et =>)
      { S7_Templates := "SrcType := Int" } GT_Contact(in1 := #iTIMER_SET, in2 := #iqTIMER_STAT)
      { S7_Templates := "SrcType := Int"; S7_GenerateENO := "TRUE" } Add(in1 := #iqTIMER_STAT, in2 := 1, out => #iqTIMER_STAT)
   END_RUNG
   // the same network as SCL:
   "trigger".TP(IN := #iENABLE AND #iPULSE, PT := T#20MS);
   IF "trigger".Q AND (#iTIMER_SET > #iqTIMER_STAT) THEN #iqTIMER_STAT := #iqTIMER_STAT + 1; END_IF;
END_REGION

REGION Network 3: if enabled and actual value equal or great than preset then OK
   RUNG wire#powerrail
      Contact( #iENABLE )
      { S7_Templates := "SrcType := Int" } LE_Contact(in1 := #iTIMER_SET, in2 := #iqTIMER_STAT)
      Coil( #tOk )
   END_RUNG
   // the same network as SCL:
   #tOk := #iENABLE AND (#iTIMER_SET <= #iqTIMER_STAT);
END_REGION

REGION Network 4: Finish
   IF #tOk THEN
       ENO := TRUE;
       RETURN;
   END_IF;
END_REGION
END_FUNCTION

FUNCTION_BLOCK "FB_IJC_AWAKE_SIGNAL"   // FB1003, LAD
TITLE = Awake signal
{ S7_Optimized_Access := 'TRUE' }
VERSION : 0.1
// This function supervise Awake signal, 
// - Awake signal is to test communication between PLC and IJCORE. 
// - Awake signal is set to 1 by PLC and set to -1 by IJCORE alternatively.
// - first PLC check if awake signal is different of 1, if it is, PLC launch timer T1 
//  (1s<T1<10s). at the end of this temporisation, PLC set awake signal to 1 and 
//  launch Timer 2. 
// - if IJCORE don't set awake signal to -1 before the end of timer 2,PLC generate  
//   Time out fault for awake signal.
// stored: AutoNumber false, IsIECCheckEnabled false, IsRetainMemResEnabled false, MemoryReserve 100, SetENOAutomatically false, UDAEnableTagReadback false
   VAR_INPUT
      ack_error : Bool;
   END_VAR
   VAR_OUTPUT
      State_com : SInt;
   END_VAR
   VAR
      T1PresetValue : Time := T#1S;
      T2PresetValue : Time := T#60S;
      AwSignalTimeOutFault : Bool := 0;
      Reset_Counters : Bool;
      Restart_Counter_bit_of_life : USInt := 0;
      NB_Bit_of_Life : Bool;
      number_restart : DInt;
      check_restart : Bool;
      "Timer" { ExternalAccessible := 'False'; ExternalVisible := 'False'; ExternalWritable := 'False'} : Array[1..5] of TON_TIME;
   END_VAR
   VAR CONSTANT
      Trestart : Time := T#200ms;
      T3 : Time := T#2s;
   END_VAR
   VAR_TEMP   // added for the SCL form of the ladder/FBD networks
      _w1 : Bool;
   END_VAR
BEGIN

REGION Network 1: - if awake signal is -1 then launch timer 1
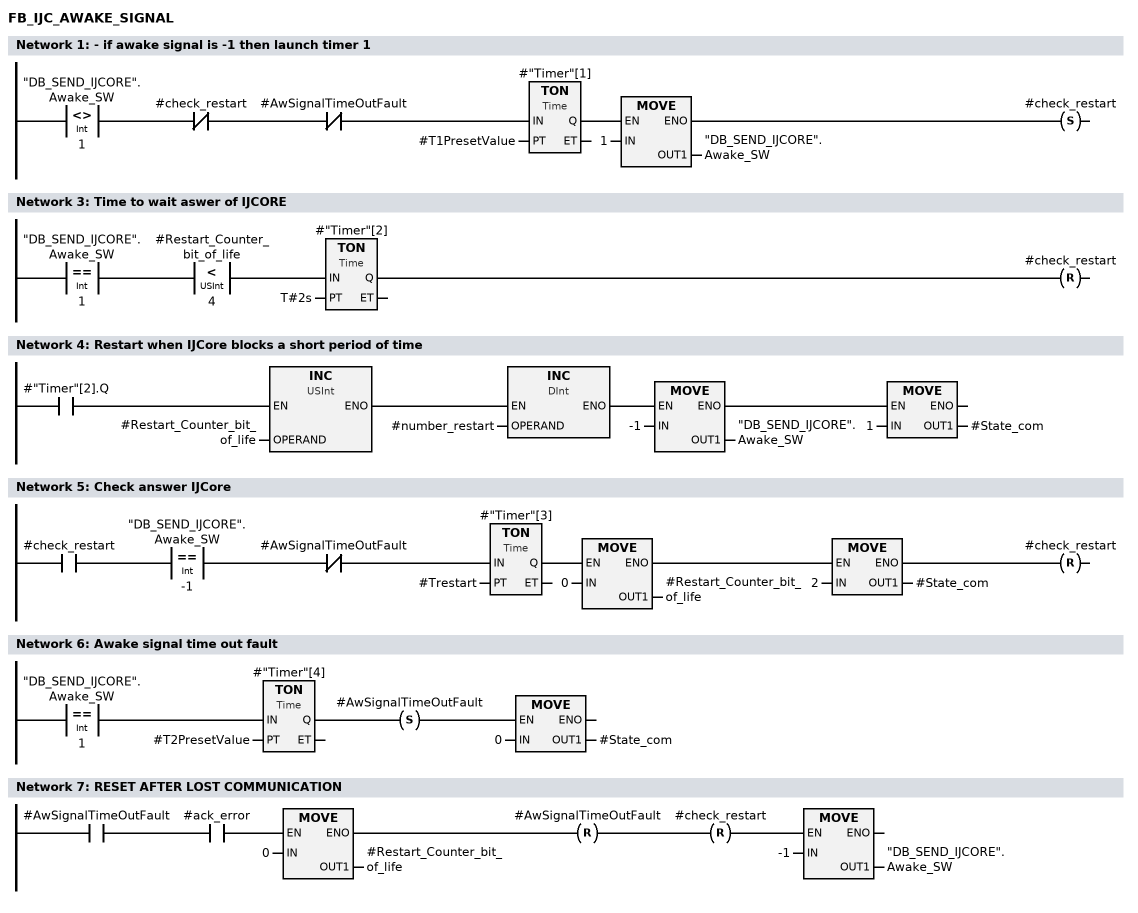
   RUNG wire#powerrail
      { S7_Templates := "SrcType := Int" } NE_Contact(in1 := "DB_SEND_IJCORE".Awake_SW, in2 := 1)
      I_Contact( #check_restart )
      I_Contact( #AwSignalTimeOutFault )
      { S7_Templates := "time_type := Time" } #"Timer"[1].TON(pt := #T1PresetValue, et =>)
      Move(in := 1, out1 => "DB_SEND_IJCORE".Awake_SW)
      S_Coil( #check_restart )
   END_RUNG
   // the same network as SCL:
   #"Timer"[1].TON(IN := ("DB_SEND_IJCORE".Awake_SW <> 1) AND NOT #check_restart AND NOT #AwSignalTimeOutFault,
                   PT := #T1PresetValue);
   IF #"Timer"[1].Q THEN
       "DB_SEND_IJCORE".Awake_SW := 1;
       #check_restart := TRUE;
   END_IF;
END_REGION

REGION Network 2: Diagnostic
END_REGION

REGION Network 3: Time to wait aswer of IJCORE
   RUNG wire#powerrail
      { S7_Templates := "SrcType := Int" } EQ_Contact(in1 := "DB_SEND_IJCORE".Awake_SW, in2 := 1)
      { S7_Templates := "SrcType := USInt" } LT_Contact(in1 := #Restart_Counter_bit_of_life, in2 := 4)
      { S7_Templates := "time_type := Time" } #"Timer"[2].TON(pt := T#2s, et =>)
      R_Coil( #check_restart )
   END_RUNG
   // the same network as SCL:
   #"Timer"[2].TON(IN := ("DB_SEND_IJCORE".Awake_SW = 1) AND (#Restart_Counter_bit_of_life < 4), PT := T#2s);
   IF #"Timer"[2].Q THEN #check_restart := FALSE; END_IF;
END_REGION

REGION Network 4: Restart when IJCore blocks a short period of time
   RUNG wire#powerrail
      Contact( #"Timer"[2].Q )
      { S7_Templates := "DestType := USInt" } Inc( #Restart_Counter_bit_of_life )
      { S7_Templates := "DestType := DInt" } Inc( #number_restart )
      Move(in := -1, out1 => "DB_SEND_IJCORE".Awake_SW)
      Move(in := 1, out1 => #State_com)
   END_RUNG
   // the same network as SCL:
   IF #"Timer"[2].Q THEN
       #Restart_Counter_bit_of_life := #Restart_Counter_bit_of_life + 1;
       #number_restart := #number_restart + 1;
       "DB_SEND_IJCORE".Awake_SW := -1;
       #State_com := 1;
   END_IF;
END_REGION

REGION Network 5: Check answer IJCore
   RUNG wire#powerrail
      Contact( #check_restart )
      { S7_Templates := "SrcType := Int" } EQ_Contact(in1 := "DB_SEND_IJCORE".Awake_SW, in2 := -1)
      I_Contact( #AwSignalTimeOutFault )
      { S7_Templates := "time_type := Time" } #"Timer"[3].TON(pt := #Trestart, et =>)
      Move(in := 0, out1 => #Restart_Counter_bit_of_life)
      Move(in := 2, out1 => #State_com)
      R_Coil( #check_restart )
   END_RUNG
   // the same network as SCL:
   #"Timer"[3].TON(IN := #check_restart AND ("DB_SEND_IJCORE".Awake_SW = (-1)) AND NOT #AwSignalTimeOutFault,
                   PT := #Trestart);
   IF #"Timer"[3].Q THEN
       #Restart_Counter_bit_of_life := 0;
       #State_com := 2;
       #check_restart := FALSE;
   END_IF;
END_REGION

REGION Network 6: Awake signal time out fault
   RUNG wire#powerrail
      { S7_Templates := "SrcType := Int" } EQ_Contact(in1 := "DB_SEND_IJCORE".Awake_SW, in2 := 1)
      { S7_Templates := "time_type := Time" } #"Timer"[4].TON(pt := #T2PresetValue, et =>)
      S_Coil( #AwSignalTimeOutFault )
      Move(in := 0, out1 => #State_com)
   END_RUNG
   // the same network as SCL:
   #"Timer"[4].TON(IN := "DB_SEND_IJCORE".Awake_SW = 1, PT := #T2PresetValue);
   IF #"Timer"[4].Q THEN
       #AwSignalTimeOutFault := TRUE;
       #State_com := 0;
   END_IF;
END_REGION

REGION Network 7: RESET AFTER LOST COMMUNICATION
   RUNG wire#powerrail
      Contact( #AwSignalTimeOutFault )
      Contact( #ack_error )
      Move(in := 0, out1 => #Restart_Counter_bit_of_life)
      R_Coil( #AwSignalTimeOutFault )
      R_Coil( #check_restart )
      Move(in := -1, out1 => "DB_SEND_IJCORE".Awake_SW)
   END_RUNG
   // the same network as SCL:
   IF #AwSignalTimeOutFault AND #ack_error THEN #Restart_Counter_bit_of_life := 0; END_IF;
   #_w1 := #AwSignalTimeOutFault AND #ack_error;
   IF #_w1 THEN
       #AwSignalTimeOutFault := FALSE;
       #check_restart := FALSE;
       "DB_SEND_IJCORE".Awake_SW := -1;
   END_IF;
END_REGION
END_FUNCTION_BLOCK

ORGANIZATION_BLOCK "stationOutputs"   // OB124, LAD, ProgramCycle
TITLE = "Main Program Sweep (Cycle)"
{ S7_Optimized_Access := 'TRUE' }
VERSION : 0.1
// stored: AutoNumber true, IsIECCheckEnabled false, SetENOAutomatically false
   VAR_INPUT
      Initial_Call : Bool;   // Initial call of this OB
      Remanence : Bool;   // =True, if remanent data are available
   END_VAR
BEGIN

REGION Network 1: PRESENT PARTS
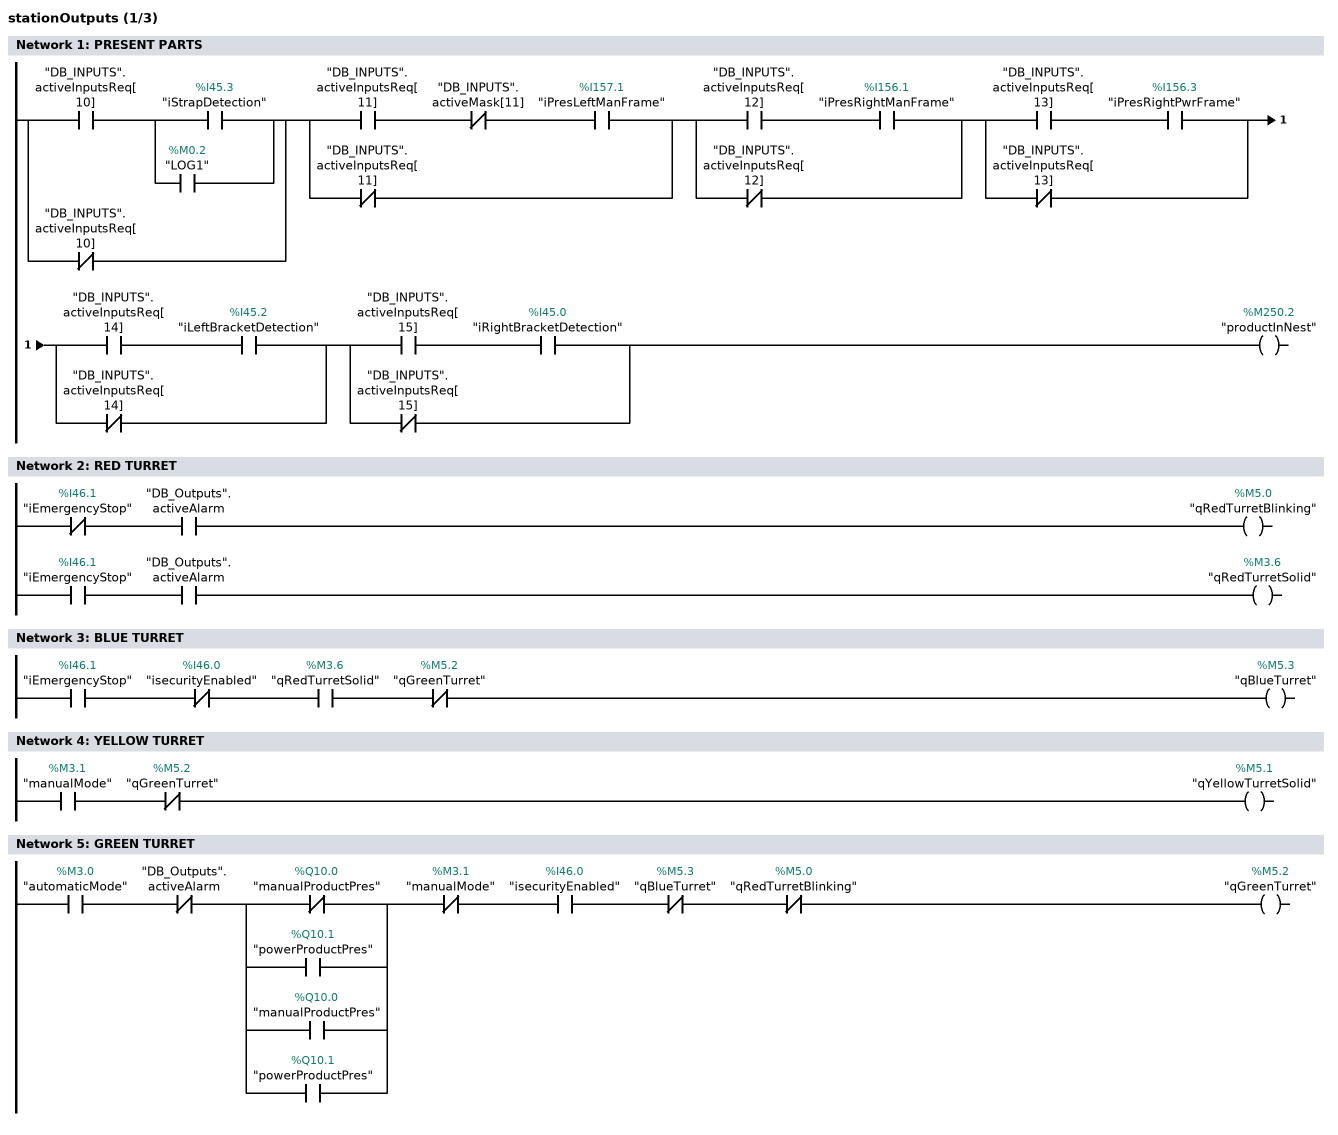
   RUNG wire#powerrail
      Contact( "DB_INPUTS".activeInputsReq[10] )
      wire#w1
      Contact( "iStrapDetection" )
      wire#w2
      Contact( "DB_INPUTS".activeInputsReq[11] )
      I_Contact( "DB_INPUTS".activeMask[11] )
      Contact( "iPresLeftManFrame" )
      wire#w3
      Contact( "DB_INPUTS".activeInputsReq[12] )
      Contact( "iPresRightManFrame" )
      wire#w4
      Contact( "DB_INPUTS".activeInputsReq[13] )
      Contact( "iPresRightPwrFrame" )
      wire#w5
      Contact( "DB_INPUTS".activeInputsReq[14] )
      Contact( "iLeftBracketDetection" )
      wire#w6
      Contact( "DB_INPUTS".activeInputsReq[15] )
      Contact( "iRightBracketDetection" )
      wire#w7
      Coil( "productInNest" )
   END_RUNG
   RUNG wire#w1
      Contact( "LOG1" )
   END_RUNG wire#w2
   RUNG wire#powerrail
      I_Contact( "DB_INPUTS".activeInputsReq[10] )
   END_RUNG wire#w2
   RUNG wire#w2
      I_Contact( "DB_INPUTS".activeInputsReq[11] )
   END_RUNG wire#w3
   RUNG wire#w3
      I_Contact( "DB_INPUTS".activeInputsReq[12] )
   END_RUNG wire#w4
   RUNG wire#w4
      I_Contact( "DB_INPUTS".activeInputsReq[13] )
   END_RUNG wire#w5
   RUNG wire#w5
      I_Contact( "DB_INPUTS".activeInputsReq[14] )
   END_RUNG wire#w6
   RUNG wire#w6
      I_Contact( "DB_INPUTS".activeInputsReq[15] )
   END_RUNG wire#w7
   // the same network as SCL:
   "productInNest" := (("DB_INPUTS".activeInputsReq[10] AND ("iStrapDetection" OR "LOG1")) OR NOT "DB_INPUTS".activeInputsReq[10]) AND (("DB_INPUTS".activeInputsReq[11] AND NOT "DB_INPUTS".activeMask[11] AND "iPresLeftManFrame") OR NOT "DB_INPUTS".activeInputsReq[11]) AND (("DB_INPUTS".activeInputsReq[12] AND "iPresRightManFrame") OR NOT "DB_INPUTS".activeInputsReq[12]) AND (("DB_INPUTS".activeInputsReq[13] AND "iPresRightPwrFrame") OR NOT "DB_INPUTS".activeInputsReq[13]) AND (("DB_INPUTS".activeInputsReq[14] AND "iLeftBracketDetection") OR NOT "DB_INPUTS".activeInputsReq[14]) AND (("DB_INPUTS".activeInputsReq[15] AND "iRightBracketDetection") OR NOT "DB_INPUTS".activeInputsReq[15]);
END_REGION

REGION Network 2: RED TURRET
   RUNG wire#powerrail
      I_Contact( "iEmergencyStop" )
      Contact( "DB_Outputs".activeAlarm )
      Coil( "qRedTurretBlinking" )
   END_RUNG
   RUNG wire#powerrail
      Contact( "iEmergencyStop" )
      Contact( "DB_Outputs".activeAlarm )
      Coil( "qRedTurretSolid" )
   END_RUNG
   // the same network as SCL:
   "qRedTurretBlinking" := NOT "iEmergencyStop" AND "DB_Outputs".activeAlarm;
   "qRedTurretSolid" := "iEmergencyStop" AND "DB_Outputs".activeAlarm;
END_REGION

REGION Network 3: BLUE TURRET
   RUNG wire#powerrail
      Contact( "iEmergencyStop" )
      I_Contact( "isecurityEnabled" )
      Contact( "qRedTurretSolid" )
      I_Contact( "qGreenTurret" )
      Coil( "qBlueTurret" )
   END_RUNG
   // the same network as SCL:
   "qBlueTurret" := "iEmergencyStop" AND NOT "isecurityEnabled" AND "qRedTurretSolid" AND NOT "qGreenTurret";
END_REGION

REGION Network 4: YELLOW TURRET
   RUNG wire#powerrail
      Contact( "manualMode" )
      I_Contact( "qGreenTurret" )
      Coil( "qYellowTurretSolid" )
   END_RUNG
   // the same network as SCL:
   "qYellowTurretSolid" := "manualMode" AND NOT "qGreenTurret";
END_REGION

REGION Network 5: GREEN TURRET
   RUNG wire#powerrail
      Contact( "automaticMode" )
      I_Contact( "DB_Outputs".activeAlarm )
      wire#w1
      I_Contact( "manualProductPres" )
      wire#w2
      I_Contact( "manualMode" )
      Contact( "isecurityEnabled" )
      I_Contact( "qBlueTurret" )
      I_Contact( "qRedTurretBlinking" )
      Coil( "qGreenTurret" )
   END_RUNG
   RUNG wire#w1
      Contact( "powerProductPres" )
   END_RUNG wire#w2
   RUNG wire#w1
      Contact( "manualProductPres" )
   END_RUNG wire#w2
   RUNG wire#w1
      Contact( "powerProductPres" )
   END_RUNG wire#w2
   // the same network as SCL:
   "qGreenTurret" := "automaticMode" AND NOT "DB_Outputs".activeAlarm AND (NOT "manualProductPres" OR "powerProductPres" OR "manualProductPres" OR "powerProductPres") AND NOT "manualMode" AND "isecurityEnabled" AND NOT "qBlueTurret" AND NOT "qRedTurretBlinking";
END_REGION

REGION Network 6: SmartLight
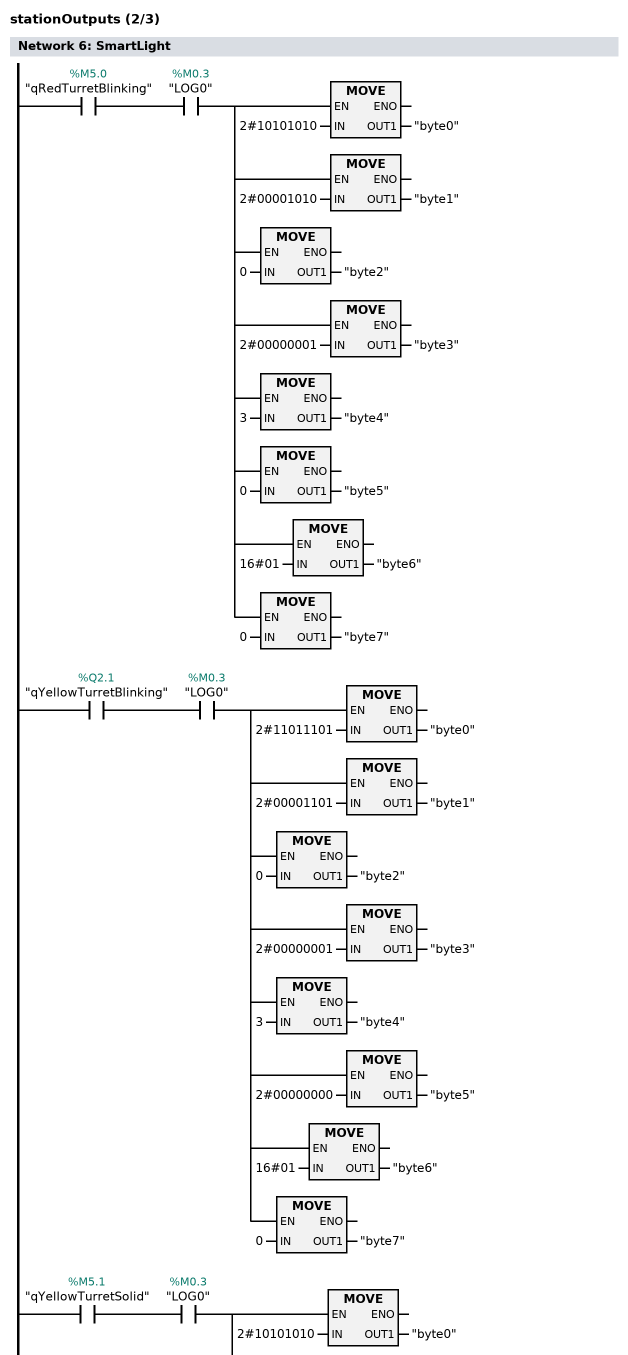
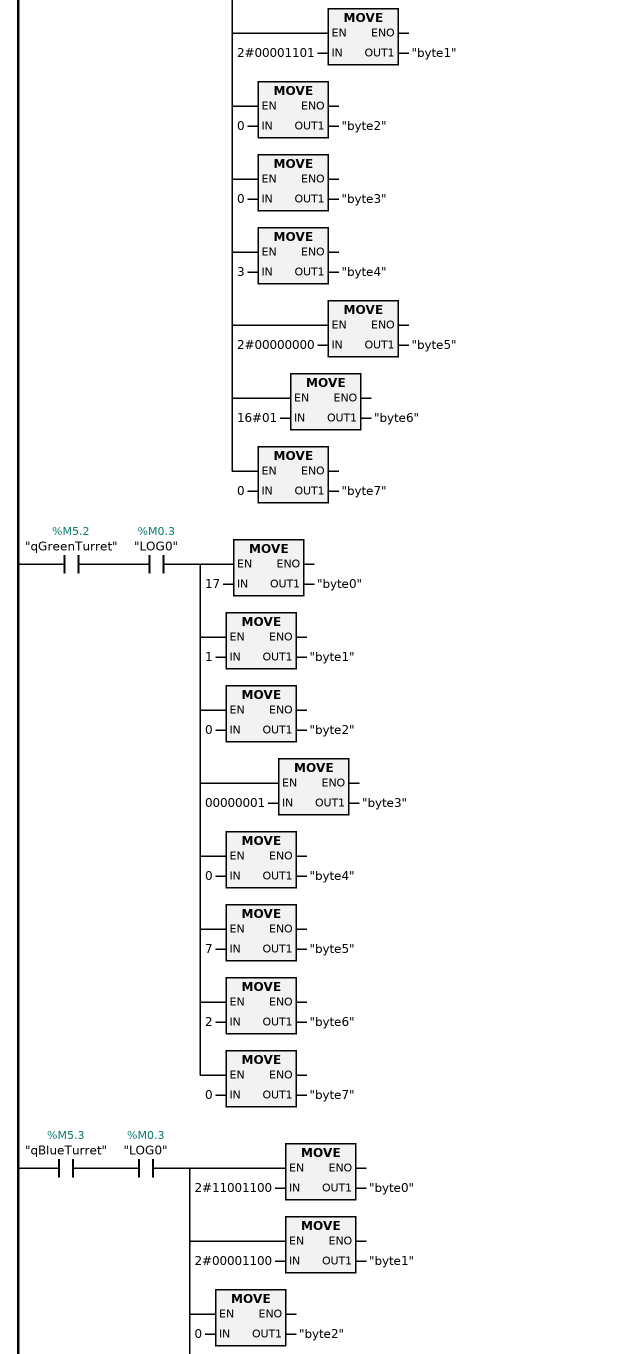
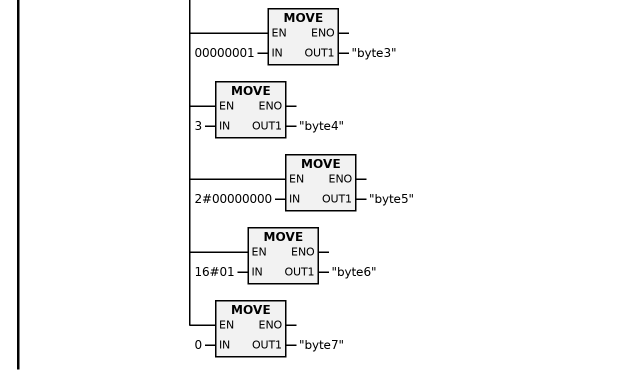
   RUNG wire#powerrail
      Contact( "qRedTurretBlinking" )
      Contact( "LOG0" )
      wire#w1
      Move(in := 2#10101010, out1 => "byte0")
   END_RUNG
   RUNG wire#w1
      Move(in := 2#00001010, out1 => "byte1")
   END_RUNG
   RUNG wire#w1
      Move(in := 0, out1 => "byte2")
   END_RUNG
   RUNG wire#w1
      Move(in := 2#00000001, out1 => "byte3")
   END_RUNG
   RUNG wire#w1
      Move(in := 3, out1 => "byte4")
   END_RUNG
   RUNG wire#w1
      Move(in := 0, out1 => "byte5")
   END_RUNG
   RUNG wire#w1
      Move(in := 16#01, out1 => "byte6")
   END_RUNG
   RUNG wire#w1
      Move(in := 0, out1 => "byte7")
   END_RUNG
   RUNG wire#powerrail
      Contact( "qYellowTurretBlinking" )
      Contact( "LOG0" )
      wire#w2
      Move(in := 2#11011101, out1 => "byte0")
   END_RUNG
   RUNG wire#w2
      Move(in := 2#00001101, out1 => "byte1")
   END_RUNG
   RUNG wire#w2
      Move(in := 0, out1 => "byte2")
   END_RUNG
   RUNG wire#w2
      Move(in := 2#00000001, out1 => "byte3")
   END_RUNG
   RUNG wire#w2
      Move(in := 3, out1 => "byte4")
   END_RUNG
   RUNG wire#w2
      Move(in := 2#00000000, out1 => "byte5")
   END_RUNG
   RUNG wire#w2
      Move(in := 16#01, out1 => "byte6")
   END_RUNG
   RUNG wire#w2
      Move(in := 0, out1 => "byte7")
   END_RUNG
   RUNG wire#powerrail
      Contact( "qYellowTurretSolid" )
      Contact( "LOG0" )
      wire#w3
      Move(in := 2#10101010, out1 => "byte0")
   END_RUNG
   RUNG wire#w3
      Move(in := 2#00001101, out1 => "byte1")
   END_RUNG
   RUNG wire#w3
      Move(in := 0, out1 => "byte2")
   END_RUNG
   RUNG wire#w3
      Move(in := 0, out1 => "byte3")
   END_RUNG
   RUNG wire#w3
      Move(in := 3, out1 => "byte4")
   END_RUNG
   RUNG wire#w3
      Move(in := 2#00000000, out1 => "byte5")
   END_RUNG
   RUNG wire#w3
      Move(in := 16#01, out1 => "byte6")
   END_RUNG
   RUNG wire#w3
      Move(in := 0, out1 => "byte7")
   END_RUNG
   RUNG wire#powerrail
      Contact( "qGreenTurret" )
      Contact( "LOG0" )
      wire#w4
      Move(in := 17, out1 => "byte0")
   END_RUNG
   RUNG wire#w4
      Move(in := 1, out1 => "byte1")
   END_RUNG
   RUNG wire#w4
      Move(in := 0, out1 => "byte2")
   END_RUNG
   RUNG wire#w4
      Move(in := 00000001, out1 => "byte3")
   END_RUNG
   RUNG wire#w4
      Move(in := 0, out1 => "byte4")
   END_RUNG
   RUNG wire#w4
      Move(in := 7, out1 => "byte5")
   END_RUNG
   RUNG wire#w4
      Move(in := 2, out1 => "byte6")
   END_RUNG
   RUNG wire#w4
      Move(in := 0, out1 => "byte7")
   END_RUNG
   RUNG wire#powerrail
      Contact( "qBlueTurret" )
      Contact( "LOG0" )
      wire#w5
      Move(in := 2#11001100, out1 => "byte0")
   END_RUNG
   RUNG wire#w5
      Move(in := 2#00001100, out1 => "byte1")
   END_RUNG
   RUNG wire#w5
      Move(in := 0, out1 => "byte2")
   END_RUNG
   RUNG wire#w5
      Move(in := 00000001, out1 => "byte3")
   END_RUNG
   RUNG wire#w5
      Move(in := 3, out1 => "byte4")
   END_RUNG
   RUNG wire#w5
      Move(in := 2#00000000, out1 => "byte5")
   END_RUNG
   RUNG wire#w5
      Move(in := 16#01, out1 => "byte6")
   END_RUNG
   RUNG wire#w5
      Move(in := 0, out1 => "byte7")
   END_RUNG
   // the same network as SCL:
   IF "qRedTurretBlinking" AND "LOG0" THEN
       "byte0" := 2#10101010;
       "byte1" := 2#00001010;
       "byte2" := 0;
       "byte3" := 2#00000001;
       "byte4" := 3;
       "byte5" := 0;
       "byte6" := 16#01;
       "byte7" := 0;
   END_IF;
   IF "qYellowTurretBlinking" AND "LOG0" THEN
       "byte0" := 2#11011101;
       "byte1" := 2#00001101;
       "byte2" := 0;
       "byte3" := 2#00000001;
       "byte4" := 3;
       "byte5" := 2#00000000;
       "byte6" := 16#01;
       "byte7" := 0;
   END_IF;
   IF "qYellowTurretSolid" AND "LOG0" THEN
       "byte0" := 2#10101010;
       "byte1" := 2#00001101;
       "byte2" := 0;
       "byte3" := 0;
       "byte4" := 3;
       "byte5" := 2#00000000;
       "byte6" := 16#01;
       "byte7" := 0;
   END_IF;
   IF "qGreenTurret" AND "LOG0" THEN
       "byte0" := 17;
       "byte1" := 1;
       "byte2" := 0;
       "byte3" := 00000001;
       "byte4" := 0;
       "byte5" := 7;
       "byte6" := 2;
       "byte7" := 0;
   END_IF;
   IF "qBlueTurret" AND "LOG0" THEN
       "byte0" := 2#11001100;
       "byte1" := 2#00001100;
       "byte2" := 0;
       "byte3" := 00000001;
       "byte4" := 3;
       "byte5" := 2#00000000;
       "byte6" := 16#01;
       "byte7" := 0;
   END_IF;
END_REGION

REGION Network 7: SMART LIGTH CONTROL
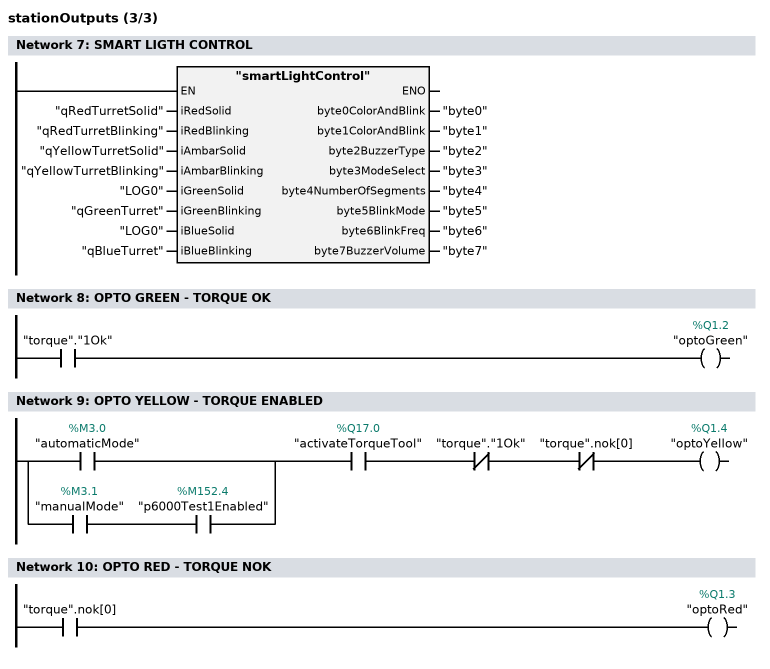
   RUNG wire#powerrail
      "smartLightControl"(iRedSolid := "qRedTurretSolid", iRedBlinking := "qRedTurretBlinking", iAmbarSolid := "qYellowTurretSolid", iAmbarBlinking := "qYellowTurretBlinking", iGreenSolid := "LOG0", iGreenBlinking := "qGreenTurret", iBlueSolid := "LOG0", iBlueBlinking := "qBlueTurret", byte0ColorAndBlink => "byte0", byte1ColorAndBlink => "byte1", byte2BuzzerType => "byte2", byte3ModeSelect => "byte3", byte4NumberOfSegments => "byte4", byte5BlinkMode => "byte5", byte6BlinkFreq => "byte6", byte7BuzzerVolume => "byte7")
   END_RUNG
   // the same network as SCL:
   "smartLightControl"(iRedSolid := "qRedTurretSolid",
                       iRedBlinking := "qRedTurretBlinking",
                       iAmbarSolid := "qYellowTurretSolid",
                       iAmbarBlinking := "qYellowTurretBlinking",
                       iGreenSolid := "LOG0",
                       iGreenBlinking := "qGreenTurret",
                       iBlueSolid := "LOG0",
                       iBlueBlinking := "qBlueTurret",
                       byte0ColorAndBlink => "byte0",
                       byte1ColorAndBlink => "byte1",
                       byte2BuzzerType => "byte2",
                       byte3ModeSelect => "byte3",
                       byte4NumberOfSegments => "byte4",
                       byte5BlinkMode => "byte5",
                       byte6BlinkFreq => "byte6",
                       byte7BuzzerVolume => "byte7");
END_REGION

REGION Network 8: OPTO GREEN - TORQUE OK
   RUNG wire#powerrail
      Contact( "torque"."1Ok" )
      Coil( "optoGreen" )
   END_RUNG
   // the same network as SCL:
   "optoGreen" := "torque"."1Ok";
END_REGION

REGION Network 9: OPTO YELLOW - TORQUE ENABLED
   RUNG wire#powerrail
      Contact( "automaticMode" )
      wire#w1
      Contact( "activateTorqueTool" )
      I_Contact( "torque"."1Ok" )
      I_Contact( "torque".nok[0] )
      Coil( "optoYellow" )
   END_RUNG
   RUNG wire#powerrail
      Contact( "manualMode" )
      Contact( "p6000Test1Enabled" )
   END_RUNG wire#w1
   // the same network as SCL:
   "optoYellow" := ("automaticMode" OR ("manualMode" AND "p6000Test1Enabled")) AND "activateTorqueTool" AND NOT "torque"."1Ok" AND NOT "torque".nok[0];
END_REGION

REGION Network 10: OPTO RED - TORQUE NOK
   RUNG wire#powerrail
      Contact( "torque".nok[0] )
      Coil( "optoRed" )
   END_RUNG
   // the same network as SCL:
   "optoRed" := "torque".nok[0];
END_REGION
END_ORGANIZATION_BLOCK

FUNCTION "smartLightControl" : Void   // FC7, LAD
{ S7_Optimized_Access := 'TRUE' }
VERSION : 0.1
// stored: AutoNumber true, IsIECCheckEnabled false, SetENOAutomatically false, UDAEnableTagReadback false
   VAR_INPUT
      iRedSolid : Bool;
      iRedBlinking : Bool;
      iAmbarSolid : Bool;
      iAmbarBlinking : Bool;
      iGreenSolid : Bool;
      iGreenBlinking : Bool;
      iBlueSolid : Bool;
      iBlueBlinking : Bool;
   END_VAR
   VAR_OUTPUT
      byte0ColorAndBlink : Byte;   // Segment 1 and 2
      byte1ColorAndBlink : Byte;   // Segment 3
      byte2BuzzerType : Byte;
      byte3ModeSelect : Byte;
      byte4NumberOfSegments : Byte;
      byte5BlinkMode : Byte;
      byte6BlinkFreq : Byte;
      byte7BuzzerVolume : Byte;
   END_VAR
   VAR_TEMP
      segment1Color : Byte;
      segment2Color : Byte;
      segment3Color : Byte;
      colorsToDisplay : Word;
      numberOfColorsToDisplay : UInt;
      colorToAddToQueue : Word;
      positionsToMove : UInt;
   END_VAR
   VAR CONSTANT
      redColor : Byte := 2#0010;
      blueColor : Byte := 2#0100;
      ambarColor : Byte := 2#0101;
      greenColor : Byte := 2#0001;
      redBlinkingColor : Byte := 2#1010;
      blueBlinkingColor : Byte := 2#1100;
      ambarBlinkingColor : Byte := 2#1101;
      greenBlinkingColor : Byte := 2#1001;
   END_VAR
BEGIN

REGION Network 1: INIT
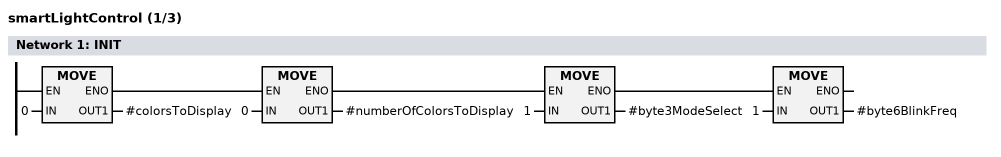
   RUNG wire#powerrail
      Move(in := 0, out1 => #colorsToDisplay)
      Move(in := 0, out1 => #numberOfColorsToDisplay)
      Move(in := 1, out1 => #byte3ModeSelect)
      Move(in := 1, out1 => #byte6BlinkFreq)
   END_RUNG
   // the same network as SCL:
   #colorsToDisplay := 0;
   #numberOfColorsToDisplay := 0;
   #byte3ModeSelect := 1;
   #byte6BlinkFreq := 1;
END_REGION

REGION Network 2: Select colors to display
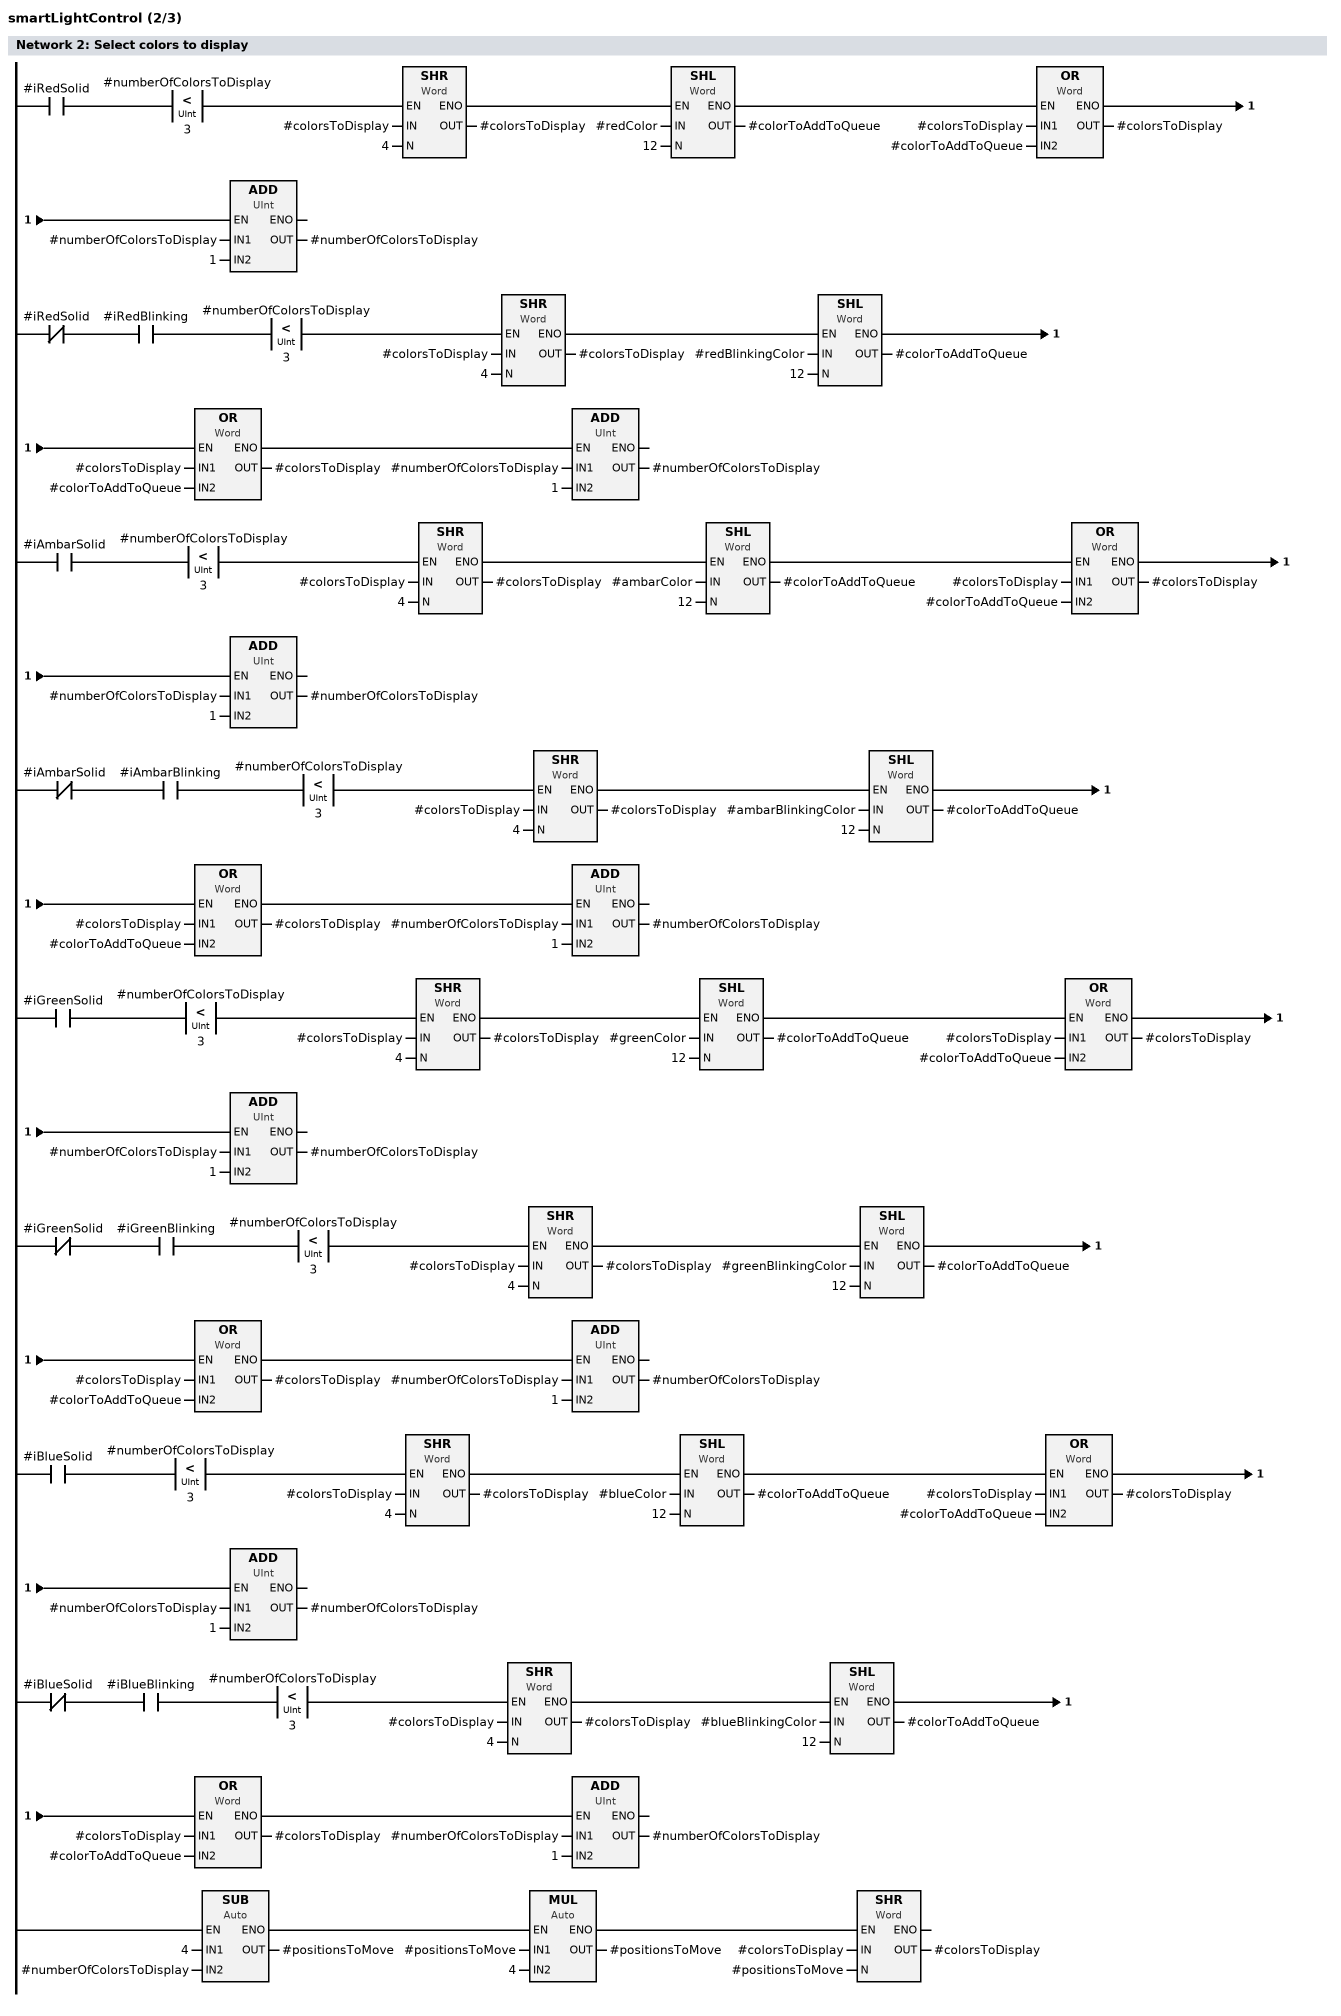
   IF #iRedSolid AND (#numberOfColorsToDisplay < 3) THEN
       #colorsToDisplay := SHR(IN := #colorsToDisplay, N := 4);
       #colorToAddToQueue := SHL(IN := #redColor, N := 12);
       #colorsToDisplay := #colorsToDisplay OR #colorToAddToQueue;
       #numberOfColorsToDisplay := #numberOfColorsToDisplay + 1;
   END_IF;
   IF NOT #iRedSolid AND #iRedBlinking AND (#numberOfColorsToDisplay < 3) THEN
       #colorsToDisplay := SHR(IN := #colorsToDisplay, N := 4);
       #colorToAddToQueue := SHL(IN := #redBlinkingColor, N := 12);
       #colorsToDisplay := #colorsToDisplay OR #colorToAddToQueue;
       #numberOfColorsToDisplay := #numberOfColorsToDisplay + 1;
   END_IF;
   IF #iAmbarSolid AND (#numberOfColorsToDisplay < 3) THEN
       #colorsToDisplay := SHR(IN := #colorsToDisplay, N := 4);
       #colorToAddToQueue := SHL(IN := #ambarColor, N := 12);
       #colorsToDisplay := #colorsToDisplay OR #colorToAddToQueue;
       #numberOfColorsToDisplay := #numberOfColorsToDisplay + 1;
   END_IF;
   IF NOT #iAmbarSolid AND #iAmbarBlinking AND (#numberOfColorsToDisplay < 3) THEN
       #colorsToDisplay := SHR(IN := #colorsToDisplay, N := 4);
       #colorToAddToQueue := SHL(IN := #ambarBlinkingColor, N := 12);
       #colorsToDisplay := #colorsToDisplay OR #colorToAddToQueue;
       #numberOfColorsToDisplay := #numberOfColorsToDisplay + 1;
   END_IF;
   IF #iGreenSolid AND (#numberOfColorsToDisplay < 3) THEN
       #colorsToDisplay := SHR(IN := #colorsToDisplay, N := 4);
       #colorToAddToQueue := SHL(IN := #greenColor, N := 12);
       #colorsToDisplay := #colorsToDisplay OR #colorToAddToQueue;
       #numberOfColorsToDisplay := #numberOfColorsToDisplay + 1;
   END_IF;
   IF NOT #iGreenSolid AND #iGreenBlinking AND (#numberOfColorsToDisplay < 3) THEN
       #colorsToDisplay := SHR(IN := #colorsToDisplay, N := 4);
       #colorToAddToQueue := SHL(IN := #greenBlinkingColor, N := 12);
       #colorsToDisplay := #colorsToDisplay OR #colorToAddToQueue;
       #numberOfColorsToDisplay := #numberOfColorsToDisplay + 1;
   END_IF;
   IF #iBlueSolid AND (#numberOfColorsToDisplay < 3) THEN
       #colorsToDisplay := SHR(IN := #colorsToDisplay, N := 4);
       #colorToAddToQueue := SHL(IN := #blueColor, N := 12);
       #colorsToDisplay := #colorsToDisplay OR #colorToAddToQueue;
       #numberOfColorsToDisplay := #numberOfColorsToDisplay + 1;
   END_IF;
   IF NOT #iBlueSolid AND #iBlueBlinking AND (#numberOfColorsToDisplay < 3) THEN
       #colorsToDisplay := SHR(IN := #colorsToDisplay, N := 4);
       #colorToAddToQueue := SHL(IN := #blueBlinkingColor, N := 12);
       #colorsToDisplay := #colorsToDisplay OR #colorToAddToQueue;
       #numberOfColorsToDisplay := #numberOfColorsToDisplay + 1;
   END_IF;
   #positionsToMove := 4 - #numberOfColorsToDisplay;
   #positionsToMove := #positionsToMove * 4;
   #colorsToDisplay := SHR(IN := #colorsToDisplay, N := #positionsToMove);
END_REGION

REGION Network 3: Send Colors to Byte 1 and 2
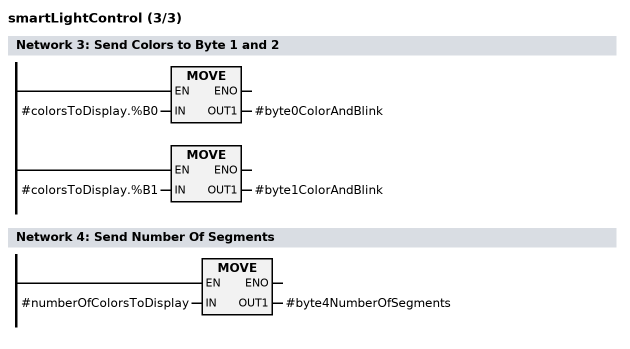
   RUNG wire#powerrail
      Move(in := #colorsToDisplay.%B0, out1 => #byte0ColorAndBlink)
   END_RUNG
   RUNG wire#powerrail
      Move(in := #colorsToDisplay.%B1, out1 => #byte1ColorAndBlink)
   END_RUNG
   // the same network as SCL:
   #byte0ColorAndBlink := #colorsToDisplay.%B0;
   #byte1ColorAndBlink := #colorsToDisplay.%B1;
END_REGION

REGION Network 4: Send Number Of Segments
   RUNG wire#powerrail
      Move(in := #numberOfColorsToDisplay, out1 => #byte4NumberOfSegments)
   END_RUNG
   // the same network as SCL:
   #byte4NumberOfSegments := #numberOfColorsToDisplay;
END_REGION
END_FUNCTION

ORGANIZATION_BLOCK "sequence"
TITLE = "Main Program Sweep (Cycle)"
{ S7_Optimized_Access := 'TRUE' }
VERSION : 0.1
   VAR_TEMP 
      i : Int;
   END_VAR


BEGIN
	IF "automaticMode" = TRUE AND "currentModel" <> 0 AND "DB_Outputs".activeAlarm =  0 THEN
	    IF "currentStep" <= "STEP".number[0] THEN
	        
	        
	//***********************************************************************************************************************************************************************           
	//***********************************************************************************************************************************************************************                  
	                                               //****ENTRADAS****//
	                                            
	                                       
	        IF ("verificacion_estados_A" = 32) THEN
	                
	            "verificacion_estados_A" := 0;
	            "a_estados" := 0;
	            "a_correctas" := 0;
	                
	          END_IF;
	        
	        
	            IF "verificacion_estados_A" <= 31 THEN
	                
	// INICIO DE CONTEO DE LOS ESTADOS_A.
	                IF "DB_INPUTS".inputActive["verificacion_estados_A"] = 1 AND "DB_INPUTS".activeInputsReq["verificacion_estados_A"] = 0 AND "DB_INPUTS".activeMask["verificacion_estados_A"] = 0 THEN
	                    "a_estados" := "a_estados" + 1;
	                END_IF;
	                
	                IF "DB_INPUTS".activeInputsReq["verificacion_estados_A"] = 0 AND "DB_INPUTS".activeMask["verificacion_estados_A"] = 1 THEN
	                    "a_estados" := "a_estados" + 1;
	                END_IF;
	                
	                IF "DB_INPUTS".activeInputsReq["verificacion_estados_A"] = 1 AND "DB_INPUTS".activeMask["verificacion_estados_A"] = 0 THEN
	                    "a_estados" := "a_estados" + 1;
	                END_IF;
	                
	                IF "DB_INPUTS".activeInputsReq["verificacion_estados_A"] = 1 AND "DB_INPUTS".activeMask["verificacion_estados_A"] = 1 THEN
	                    "a_estados" := "a_estados" + 1;
	                END_IF;
	// INICIO DE CONTEO DE TODOS LOS ESTADOS_A.
	                
	// INICIO DE CONTEO DE ESTADO DE ENTRADAS CORRECTAS.
	                IF "DB_INPUTS".inputActive["verificacion_estados_A"] = 0 AND "DB_INPUTS".activeInputsReq["verificacion_estados_A"] = 0 AND "DB_INPUTS".activeMask["verificacion_estados_A"] = 1 THEN
	                    "a_correctas" := "a_correctas" + 1;
	                END_IF;
	                
	                IF "DB_INPUTS".inputActive["verificacion_estados_A"] = 0 AND "DB_INPUTS".activeInputsReq["verificacion_estados_A"] = 1 AND "DB_INPUTS".activeMask["verificacion_estados_A"] = 1 THEN
	                    "a_correctas" := "a_correctas" + 1;
	                END_IF;
	                
	                IF "DB_INPUTS".inputActive["verificacion_estados_A"] = 1 AND "DB_INPUTS".activeInputsReq["verificacion_estados_A"] = 0 AND "DB_INPUTS".activeMask["verificacion_estados_A"] = 1 THEN
	                    "a_correctas" := "a_correctas" + 1;
	                END_IF;
	                
	                IF "DB_INPUTS".inputActive["verificacion_estados_A"] = 1 AND "DB_INPUTS".activeInputsReq["verificacion_estados_A"] = 1 AND "DB_INPUTS".activeMask["verificacion_estados_A"] = 0 THEN
	                    "a_correctas" := "a_correctas" + 1;
	                END_IF;
	                
	                IF "DB_INPUTS".inputActive["verificacion_estados_A"] = 1 AND "DB_INPUTS".activeInputsReq["verificacion_estados_A"] = 1 AND "DB_INPUTS".activeMask["verificacion_estados_A"] = 1 THEN
	                    "a_correctas" := "a_correctas" + 1;
	                END_IF;
	// FIN DE CONTEO DE ESTADO DE ENTRADAS CORRECTAS.
	                
	                "verificacion_estados_A" := "verificacion_estados_A" + 1;
	            END_IF;
	            
	            
	//***********************************************************************************************************************************************************************           
	//***********************************************************************************************************************************************************************                  
	                                                        //****SALIDAS****//         
	                                                        
	            IF "verificacion_estados_B" = 32 THEN
	                
	                "verificacion_estados_B" := 0;
	                "b_estados" := 0;
	                "numberOfCorrectOutputStates" := 0;
	                
	            END_IF;
	            
	            IF "verificacion_estados_B" <= 31 THEN
	                
	// INICIO DE CONTEO DE LOS ESTADOS_B.
	                IF "DB_Outputs".outputsActive["verificacion_estados_B"] = 1 AND "DB_Outputs".activeOutputsReq["verificacion_estados_B"] = 0 AND "DB_Outputs".activeMask["verificacion_estados_B"] = 0 THEN
	                    "b_estados" := "b_estados" + 1;
	                END_IF;
	                
	                IF "DB_Outputs".activeOutputsReq["verificacion_estados_B"] = 0 AND "DB_Outputs".activeMask["verificacion_estados_B"] = 1 THEN
	                    "b_estados" := "b_estados" + 1;
	                END_IF;
	                
	                IF "DB_Outputs".activeOutputsReq["verificacion_estados_B"] = 1 AND "DB_Outputs".activeMask["verificacion_estados_B"] = 0 THEN
	                    "b_estados" := "b_estados" + 1;
	                END_IF;
	                
	                IF "DB_Outputs".activeOutputsReq["verificacion_estados_B"] = 1 AND "DB_Outputs".activeMask["verificacion_estados_B"] = 1 THEN
	                    "b_estados" := "b_estados" + 1;
	                END_IF;
	// FIN DE CONTEO DE TODOS LOS ESTADOS_B.
	                
	                
	// DESACTIVACIÓN DE SALIDA CUANDO NO ES REQUERIDA.
	                
	                IF "DB_Outputs".activeOutputsReq["verificacion_estados_B"] = 0 THEN
	                    "DB_Outputs".activateOutput["verificacion_estados_B"] := 0;
	                END_IF;
	                
	            
	// INICIO DE CONTEO DE ESTADO DE "SALIDAS" CORRECTAS.
	                IF "DB_Outputs".activeOutputsReq["verificacion_estados_B"] = 0 AND "DB_Outputs".activeMask["verificacion_estados_B"] = 1 THEN
	                    "numberOfCorrectOutputStates" := "numberOfCorrectOutputStates" + 1;
	                  
	                END_IF;
	                
	                IF "DB_Outputs".activeOutputsReq["verificacion_estados_B"] = 1 AND "DB_Outputs".activeMask["verificacion_estados_B"] = 1 THEN
	                    "DB_Outputs".activateOutput["verificacion_estados_B"] := 1;
	                    //IF "SALIDAS".TIMER ["verificacion_estados_B"].Q = 1 THEN
	                        "numberOfCorrectOutputStates" := "numberOfCorrectOutputStates" + 1;
	                    // END_IF;
	                END_IF;
	                
	                IF "DB_Outputs".activeOutputsReq["verificacion_estados_B"] = 1 AND "DB_Outputs".activeMask["verificacion_estados_B"] = 0 THEN
	                    "DB_Outputs".activateOutput["verificacion_estados_B"] := 1;
	                   // IF "SALIDAS".TIMER ["verificacion_estados_B"].Q = 1 THEN
	                        IF "DB_Outputs".outputsActive["verificacion_estados_B"] = 1 THEN
	                            "numberOfCorrectOutputStates" := "numberOfCorrectOutputStates" + 1;
	                        END_IF;
	                   //END_IF;
	                END_IF;
	                
	// FIN DE CONTEO DE ESTADO DE "SALIDAS" CORRECTAS.
	                
	                "verificacion_estados_B" := "verificacion_estados_B" + 1;
	            END_IF;
	            
	            
	                                                     
	//***********************************************************************************************************************************************************************           
	//***********************************************************************************************************************************************************************                  
	                                                     //****ENTRADAS****//
	                                                     
	            IF "DB_Outputs".showTextOutPuts = 0 THEN
	                
	                IF "aa" <= 31 THEN
	                    
	// INICIO DE COMPARACIONES DE DETECCIÓN DE SEÑALES DE ENTRADAS FALTANTES O SOBRANTES.  
	                    IF ("DB_INPUTS".activeMask["aa"] = 1) OR (("DB_INPUTS".activeInputsReq["aa"] = 1) AND ("DB_INPUTS".inputActive["aa"] = 1)) OR (("DB_INPUTS".activeInputsReq["aa"] = 0) AND ("DB_INPUTS".inputActive["aa"] = 0)) THEN
	                        "aa" := "aa" + 1;
	                        IF "aa" = 32 THEN
	                            "aa" := 0;
	                            "DB_Outputs".showTextOutPuts := 1;
	                        END_IF;
	                    END_IF;
	                    
	                    IF ("DB_INPUTS".activeMask["aa"] = 0) AND "DB_INPUTS".activeInputsReq["aa"] = 1 AND "DB_INPUTS".inputActive["aa"] = 0 THEN
	                        
	                        IF "allowedTextChange" = 0 THEN
	                            "DB_HMI".operatorTextIndicator := CONCAT(IN1 := 'ESPERANDO POR ', IN2 := "DB_INPUTS".inputText["aa"]);
	                            "aa" := "aa" + 1;
	                            IF "aa" = 32 THEN
	                                "aa" := 0;
	                                "DB_Outputs".showTextOutPuts := 1;
	                            END_IF;
	                        END_IF;
	                        
	                    END_IF;
	                    
	                    IF ("DB_INPUTS".activeMask["aa"] = 0) AND "DB_INPUTS".activeInputsReq["aa"] = 0 AND "DB_INPUTS".inputActive["aa"] = 1 THEN
	                        
	                        IF "allowedTextChange" = 0 THEN
	                            "DB_HMI".operatorTextIndicator := CONCAT(IN1 := 'ESPERANDO POR NO ', IN2 := "DB_INPUTS".inputText["aa"]);
	                            "aa" := "aa" + 1;
	                            IF "aa" = 32 THEN
	                                "aa" := 0;
	                                "DB_Outputs".showTextOutPuts := 1;
	                            END_IF;
	                        END_IF;
	                        
	                    END_IF;
	//FIN DE COMPARACIONES DE DETECCIÓN DE SEÑALES DE ENTRADAS FALTANTES O SOBRANTES. 
	                    
	                    
	                END_IF;
	            END_IF;
	            
	        
	        
	//***********************************************************************************************************************************************************************           
	//***********************************************************************************************************************************************************************                  
	                                                    //****SALIDAS****//
	                                                   
	            IF "DB_Outputs".showTextOutPuts = 1 THEN
	                
	                IF "bb" <= 31 THEN
	                    
	// INICIO DE COMPARACIONES DE DETECCIÓN DE SEÑALES DE SALIDAS FALTANTES O SOBRANTES.  
	                    IF ("DB_Outputs".activeMask["bb"] = 1) OR (("DB_Outputs".activeOutputsReq["bb"] = 1) AND ("DB_Outputs".outputsActive["bb"] = 1)) OR (("DB_Outputs".activeOutputsReq["bb"] = 0) AND ("DB_Outputs".outputsActive["bb"] = 0)) THEN
	                        "bb" := "bb" + 1;
	                        IF "bb" = 32 THEN
	                           "bb" := 0;
	                           "DB_Outputs".showTextOutPuts := 0;
	                        END_IF;
	                    END_IF;
	                    
	                    IF ("DB_Outputs".activeMask["bb"] = 0) AND "DB_Outputs".activeOutputsReq["bb"] = 1 AND "DB_Outputs".outputsActive["bb"] = 0 THEN
	                        
	                        IF "allowedTextChange" = 0 THEN
	                            "DB_HMI".operatorTextIndicator := CONCAT(IN1 := 'ESPERANDO POR ', IN2 := "DB_Outputs".text["bb"]);
	                            "bb" := "bb" + 1;
	                            IF "bb" = 32 THEN
	                                "bb" := 0;
	                                "DB_Outputs".showTextOutPuts := 0;
	                            END_IF;
	                        END_IF;
	                        
	                    END_IF;
	                    
	                    IF ("DB_Outputs".activeMask["bb"] = 0) AND "DB_Outputs".activeOutputsReq["bb"] = 0 AND "DB_Outputs".outputsActive["bb"] = 1 THEN
	                        
	                        IF "allowedTextChange" = 0 THEN
	                            "DB_HMI".operatorTextIndicator := CONCAT(IN1 := 'ESPERANDO POR NO ', IN2 := "DB_Outputs".text["bb"]);
	                            "bb" := "bb" + 1;
	                            IF "bb" = 32 THEN
	                                "bb" := 0;
	                                "DB_Outputs".showTextOutPuts := 0;
	                            END_IF;
	                        END_IF;
	                        
	                    END_IF;
	// FIN DE COMPARACIONES DE DETECCIÓN DE SEÑALES DE SALIDAS FALTANTES O SOBRANTES. 
	
	                END_IF;
	            END_IF;
	                                                    
	                                                    
	                                                    
	//***********************************************************************************************************************************************************************           
	//***********************************************************************************************************************************************************************                  
	                                                    //****CAMBIO DE PASO****//
	                                                    
	                                                    
	               
	            IF (("a_correctas" = "a_estados") AND ("a_correctas" <> 0) AND ("a_estados" <> 0) AND ("numberOfCorrectOutputStates" = "b_estados") AND ("numberOfCorrectOutputStates" <> 0) AND ("b_estados" <> 0) AND ("verificacion_estados_B" = 32) AND ("verificacion_estados_A" = 32)) OR (("DB_INPUTS".intputSequence[0, "currentStep"] = 0) AND ("DB_INPUTS".maskSequence[0, "currentStep"] = 0) AND ("DB_INPUTS".activeInputsReqDInt = 0) AND ("verificacion_estados_A" = 32)) OR (("a_correctas" = "a_estados") AND ("a_correctas" <> 0) AND ("a_estados" <> 0) AND ("verificacion_estados_A" = 32) AND ("DB_Outputs".outputSequence[0, "currentStep"] = 0) AND ("DB_Outputs".maskSequence[0, "currentStep"] = 0) AND ("DB_Outputs".active = 0)) THEN
	                
	                "DB_HMI".operatorTextIndicator := ' ';
	                
	                "STEP".stepChangeTimerStart := 1;
	                
	                IF "STEP".counterDone = 1 THEN
	                    "STEP".stepChangeTimerStart := 0;
	                END_IF;
	                
	                IF ("STEP".counterDone = 1 OR "STEP".stepChangeTimer = 0) THEN
	                    
	                    IF "currentStep" = "STEP".number[0] THEN
	                        IF "currentStep" <> 0 AND "STEP".number[0] <> 0 THEN
	                            "DB_HMI".cicles := "DB_HMI".cicles + 1;
	                            
	                            IF "shift1" THEN
	                                "DB_HMI".production1 := "DB_HMI".production1 + 1;
	                            END_IF;
	                            
	                            IF "shift2" THEN
	                                "DB_HMI".production2 := "DB_HMI".production2 + 1;
	                            END_IF;
	                            
	                            IF "shift3" THEN
	                                "DB_HMI".production3 := "DB_HMI".production3 + 1;
	                            END_IF;
	                            
	                            
	                        END_IF;
	                        "currentStep" := 0;
	                        RETURN;
	                    END_IF;
	                    
	                    "currentStep" := "currentStep" + 1;
	                   
	                END_IF;
	                
	                
	            END_IF;
	            
	            
	            
	        END_IF;
	      END_IF;
	      
	      
END_ORGANIZATION_BLOCK

FUNCTION "FC_TRACE_TRR" : Void
{ S7_Optimized_Access := 'TRUE' }
VERSION : 0.1
   VAR_INPUT 
      Req : Bool;   // Request message
      MessageNumber : DInt;   // Message number
      TraceabilityMode : Int;   // Tracability mode
      NFP : String;
      ProcessStatus : USInt;
      NumberOfProcess : USInt;
      ErrReset : Bool;
   END_VAR

   VAR_OUTPUT 
      MessageDone : Bool;
      Answer : Int;
   END_VAR

   VAR_IN_OUT 
      State : USInt;
   END_VAR

   VAR_TEMP 
      SEND_OFFSET : Struct
         SW : DInt;
         MSG : DInt;
      END_STRUCT;
      REC_OFFSET : Struct
         SW : DInt;
         MSG : DInt;
         ANS : DInt;
      END_STRUCT;
      IDB : Int;
      i : Int;
      j : Int;
      k : Int;
      CNT : Int;
      CNT_STR : String[2];
      MSG : DInt;
      ErrCode : Int;
   END_VAR

   VAR CONSTANT 
      "DB" : Byte := 16#84;
      CLEAR : Word := 16#0000;
      MINUS1 : Word := 16#FFFF;
      PLUS1 : Word := 16#0001;
      DB_REC : DB_ANY := 1006;
      DB_SEND : DB_ANY := 1005;
      Blank : String := '';
   END_VAR


BEGIN
	//TITLE = 'IJCORE PROTOCOL'
	//AUTHOR: RAUL ROBINS
	//CREATED ON: 03/24/2023
	//VERSION: 3.0
	
	
	
	IF #MessageNumber < 1  THEN
	    RETURN;
	END_IF;
	
	
	
	
	IF NOT #Req THEN // Error Reset
	    #State := 0;
	END_IF;
	
	#SEND_OFFSET.SW := (#MessageNumber * 2) + 2; //Calc message send sw offset
	#SEND_OFFSET.MSG := ((#MessageNumber - 1) * 80) + 604; // Calc send message offset
	#REC_OFFSET.SW := (#MessageNumber - 1) * 2; // Calc receive sw offset
	#REC_OFFSET.ANS := ((#MessageNumber - 1) * 32) + 600; // Calc receive answer offset
	#REC_OFFSET.MSG := ((#MessageNumber - 1) * 32) + 602; // Calc receive message offset
	
	
	CASE #State OF
	    0: // Initial State
	        #MessageDone := FALSE;
	        #Answer := 0;
	
	        POKE(area := #DB, //Clear send flag
	             dbNumber := #DB_SEND,
	             byteOffset := #SEND_OFFSET.SW,
	             value := #MINUS1);
	        POKE(area := #DB, //Clear receive flag
	             dbNumber := #DB_REC,
	             byteOffset := #REC_OFFSET.SW,
	             value := #MINUS1);
	     
	        #State := 10; ///Transition to state 10
	        
	    10: // Wait for start command
	        IF #Req AND
	            #ProcessStatus > 0  THEN //If start command active
	            
	            POKE(area := #DB, //Clear send flag
	                 dbNumber := #DB_SEND,
	                 byteOffset := #SEND_OFFSET.SW,
	                 value := #MINUS1);
	            POKE(area := #DB, //Clear receive flag
	                 dbNumber := #DB_REC,
	                 byteOffset := #REC_OFFSET.SW,
	                 value := #MINUS1);
	            POKE(area := #DB, // Clear answer 
	                 dbNumber := #DB_REC,
	                 byteOffset := #REC_OFFSET.ANS,
	                 value := #CLEAR);
	            
	            FOR #i := 0 TO 79 BY 1 DO //Clear all send array
	                POKE(area := #DB,
	                     dbNumber := #DB_SEND,
	                     byteOffset := (#SEND_OFFSET.MSG + #i),
	                     value := '$00');
	            END_FOR;
	            FOR #i := 0 TO 29 BY 1 DO //Clear all receive array
	                POKE(area := #DB,
	                     dbNumber := #DB_REC,
	                     byteOffset := (#REC_OFFSET.MSG + #i),
	                     value := '$00');
	            END_FOR;
	            #State := 20; //Transition to state 20
	        END_IF;
	        
	    20: // Create message to send
	        FOR #i := 0 TO 7 BY 1 DO //Copy NFP to DB to send
	            POKE(area := #DB,
	                 dbNumber := #DB_SEND,
	                 byteOffset := (#SEND_OFFSET.MSG + #i),
	                 value := #NFP[#i + 1]);
	        END_FOR;
	                
	  
	                
	                POKE(area := #DB, //Set the process status of the message
	                     dbNumber := #DB_SEND,
	                     byteOffset := (#SEND_OFFSET.MSG + 8),
	                     value := USINT_TO_CHAR(#ProcessStatus + 48));
	                
	          
	        #State := 30; // Transition to state 30
	        
	    30: //Set flag to "1" to inform that PLC is ready to send (DB5 Ó 1005)
	        POKE(area := #DB,//Set flag to "1" to inform that PLC is ready to send
	             dbNumber := #DB_SEND,
	             byteOffset := #SEND_OFFSET.SW,
	             value := #PLUS1);
	        #State := 40; // Transition to state 40
	        
	        
	    40: //Wait to IJCORE response with "-1"
	        IF (PEEK_WORD(area := #DB, dbNumber := #DB_SEND, byteOffset := #SEND_OFFSET.SW) = #MINUS1)
	        THEN
	            #State := 50; // Transition to state 50
	        END_IF;
	        
	    50: //Check if IJCORE have answer from DB Receive
	        IF (PEEK_WORD(area := #DB, dbNumber := #DB_REC, byteOffset := #REC_OFFSET.SW) = #PLUS1)
	        THEN
	            #Answer := WORD_TO_INT(PEEK_WORD(area := #DB, dbNumber := #DB_REC, byteOffset := #REC_OFFSET.ANS)); //Copy answer from IJCORE
	
	            #State := 60; // Transition to state 100
	        END_IF;
	        
	    60: //Change Flag to "-1"
	        POKE(area := #DB, //Set "-1" to IJCORE
	             dbNumber := #DB_REC,
	             byteOffset := #REC_OFFSET.SW,
	             value := #MINUS1);
	        #State := 100; // Transition to state 100
	        
	        
	    100: //Sequence done
	        CASE #TraceabilityMode OF
	            1:// Full traceability
	                IF #Answer = 1 THEN
	                    #MessageDone := TRUE;
	                ELSE
	                    #MessageDone := FALSE;
	                END_IF;
	            2:// Traceability only
	                #MessageDone := TRUE;
	        END_CASE;
	        
	        IF NOT #Req THEN
	            #State := 0; // Transition to state 0
	        END_IF;
	END_CASE;
	
	
	
	
	
	
	
END_FUNCTION

FUNCTION "FC_READING_IJC_TRS" : Void
{ S7_Optimized_Access := 'TRUE' }
VERSION : 0.1
   VAR_INPUT 
      Req : Bool;   // Request message
      MessageNumber : DInt;   // Message number
      TraceabilityMode : Int;   // Tracability mode
      NFP : String;   // NFP
      ProcessStatus : UInt;   // Process status
      ScrewData : "UDT_ScrewData";   // Screw data
      ErrReset : Bool;   // Error reset
   END_VAR

   VAR_OUTPUT 
      MessageDone : Bool;   // Mesagge Complete
   END_VAR

   VAR_IN_OUT 
      Answer : Int;   // Answer from ijcore
      State : USInt;   // s
   END_VAR

   VAR_TEMP 
      SEND_OFFSET : Struct
         SW : DInt;
         MSG : DInt;
      END_STRUCT;
      REC_OFFSET : Struct
         SW : DInt;
         MSG : DInt;
         ANS : DInt;
      END_STRUCT;
      IDB : Int;
      i : Int;
      j : Int;
      k : Int;
      MSG : DInt;
      ErrCode : Int;
      CNT : Int;
      CNT_STR : String[2];
   END_VAR

   VAR CONSTANT 
      "DB" : Byte := 16#84;
      CLEAR : Word := 16#0000;
      MINUS1 : Word := 16#FFFF;
      PLUS1 : Word := 16#0001;
      DB_REC : DB_ANY := 1006;
      DB_SEND : DB_ANY := 1005;
      Blank : String := '';
   END_VAR


BEGIN
	//TITLE = 'IJCORE PROTOCOL TRS'
	//AUTHOR: RAUL ROBINS
	//CREATED ON: 03/24/2023
	//VERSION: 3.0
	
	
	
	IF #MessageNumber < 1  THEN
	    RETURN;
	END_IF;
	
	
	
	
	IF NOT #Req THEN // Error Reset
	    #State := 0;
	END_IF;
	
	#SEND_OFFSET.SW := (#MessageNumber * 2) + 2; //Calc message send sw offset
	#SEND_OFFSET.MSG := ((#MessageNumber - 1) * 80) + 604; // Calc send message offset
	#REC_OFFSET.SW := (#MessageNumber - 1) * 2; // Calc receive sw offset
	#REC_OFFSET.ANS := ((#MessageNumber - 1) * 32) + 600; // Calc receive answer offset
	#REC_OFFSET.MSG := ((#MessageNumber - 1) * 32) + 602; // Calc receive message offset
	
	
	CASE #State OF
	    0: // Initial State
	        #MessageDone := FALSE;
	        #Answer := 0;
	
	        POKE(area := #DB, //Clear send flag
	             dbNumber := #DB_SEND,
	             byteOffset := #SEND_OFFSET.SW,
	             value := #MINUS1);
	        POKE(area := #DB, //Clear receive flag
	             dbNumber := #DB_REC,
	             byteOffset := #REC_OFFSET.SW,
	             value := #MINUS1);
	     
	        #State := 10; ///Transition to state 10
	        
	    10: // Wait for start command
	        IF #Req THEN //If start command active
	            
	            POKE(area := #DB, //Clear send flag
	                 dbNumber := #DB_SEND,
	                 byteOffset := #SEND_OFFSET.SW,
	                 value := #MINUS1);
	            POKE(area := #DB, //Clear receive flag
	                 dbNumber := #DB_REC,
	                 byteOffset := #REC_OFFSET.SW,
	                 value := #MINUS1);
	            POKE(area := #DB, // Clear answer 
	                 dbNumber := #DB_REC,
	                 byteOffset := #REC_OFFSET.ANS,
	                 value := #CLEAR);
	            
	            FOR #i := 0 TO 79 BY 1 DO //Clear all send array
	                POKE(area := #DB,
	                     dbNumber := #DB_SEND,
	                     byteOffset := (#SEND_OFFSET.MSG + #i),
	                     value := '$00');
	            END_FOR;
	            FOR #i := 0 TO 29 BY 1 DO //Clear all receive array
	                POKE(area := #DB,
	                     dbNumber := #DB_REC,
	                     byteOffset := (#REC_OFFSET.MSG + #i),
	                     value := '$00');
	            END_FOR;
	            #State := 20; //Transition to state 20
	        END_IF;
	        
	    20: // Create message to send
	        FOR #i := 0 TO 7 BY 1 DO //Copy NFP to DB to send
	            POKE(area := #DB,
	                 dbNumber := #DB_SEND,
	                 byteOffset := (#SEND_OFFSET.MSG + #i),
	                 value := #NFP[#i + 1]);
	        END_FOR;
	        //Copy process status 
	        POKE(area := #DB,
	             dbNumber := #DB_SEND,
	             byteOffset := (#SEND_OFFSET.MSG + 8),
	             value := #ProcessStatus);
	        //Copy toque and angle 
	        POKE(area := #DB,
	             dbNumber := #DB_SEND,
	             byteOffset := (#SEND_OFFSET.MSG + 9),
	             value := BYTE_TO_CHAR(49));
	        //ANGLE
	        POKE(area := #DB,
	             dbNumber := #DB_SEND,
	             byteOffset := (#SEND_OFFSET.MSG + 10),
	             value := #ScrewData.Angle);
	        //TORQUE BEFORE POINT
	        POKE(area := #DB,
	             dbNumber := #DB_SEND,
	             byteOffset := (#SEND_OFFSET.MSG + #k + 11),
	             value := #ScrewData.Torque.BeforePoint);
	        
	        //TORQUE AFTER POINT
	        POKE(area := #DB,
	             dbNumber := #DB_SEND,
	             byteOffset := (#SEND_OFFSET.MSG + #k + 12),
	             value := #ScrewData.Torque.AfterPoint);
	        
	        #State := 30; // Transition to state 30
	        
	    30: //Set flag to "1" to inform that PLC is ready to send (DB5 Ó 1005)
	        POKE(area := #DB,//Set flag to "1" to inform that PLC is ready to send
	             dbNumber := #DB_SEND,
	             byteOffset := #SEND_OFFSET.SW,
	             value := #PLUS1);
	        #State := 40; // Transition to state 40
	        
	        
	    40: //Wait to IJCORE response with "-1"
	        IF (PEEK_WORD(area := #DB, dbNumber := #DB_SEND, byteOffset := #SEND_OFFSET.SW) = #MINUS1)
	        THEN
	            #State := 50; // Transition to state 50
	        END_IF;
	        
	    50: //Check if IJCORE have answer from DB Receive
	        IF (PEEK_WORD(area := #DB, dbNumber := #DB_REC, byteOffset := #REC_OFFSET.SW) = #PLUS1)
	        THEN
	            #Answer := WORD_TO_INT(PEEK_WORD(area := #DB, dbNumber := #DB_REC, byteOffset := #REC_OFFSET.ANS)); //Copy answer from IJCORE
	            //Ensure aswer is copied
	            IF #Answer <> 0 THEN
	                #State := 60; // Transition to state 100
	            END_IF;
	        END_IF;
	        
	    60: //Change Flag to "-1"
	        POKE(area := #DB, //Set "-1" to IJCORE
	             dbNumber := #DB_REC,
	             byteOffset := #REC_OFFSET.SW,
	             value := #MINUS1);
	        #State := 100; // Transition to state 100
	        
	        
	    100: //Sequence done
	        CASE #TraceabilityMode OF
	            1:// Full traceability
	                IF #Answer = 1 THEN
	                    #MessageDone := TRUE;
	                ELSE
	                    #MessageDone := FALSE;
	                END_IF;
	            2:// Traceability only
	                #MessageDone := TRUE;
	        END_CASE;
	        
	        IF NOT #Req THEN
	            #State := 0; // Transition to state 0
	        END_IF;
	END_CASE;
	
	
	
	
	
	
	
END_FUNCTION

DATA_BLOCK "BUTTON SHUTOFF TIME"   // DB8
{ S7_Optimized_Access := 'TRUE' }
// stored: AutoNumber true, DBAccessibleFromOPCUA true, DBAccessibleFromWebserver true, InstanceOfName IEC_TIMER, OfSystemLibElement IEC_TIMER, OfSystemLibVersion 1.0
"IEC_TIMER"
   // VAR
   //    PT : Time := T#0MS;
   //    ET { ExternalWritable := 'False'} : Time;
   //    IN : Bool := FALSE;
   //    Q { ExternalWritable := 'False'} : Bool;
   // END_VAR
BEGIN
END_DATA_BLOCK

DATA_BLOCK "CYL 10 DIR A TON"   // DB50
{ S7_Optimized_Access := 'TRUE' }
// stored: AutoNumber true, DBAccessibleFromOPCUA true, DBAccessibleFromWebserver true, InstanceOfName IEC_TIMER, OfSystemLibElement IEC_TIMER, OfSystemLibVersion 1.0
"IEC_TIMER"
   // VAR
   //    PT : Time := T#0MS;
   //    ET { ExternalWritable := 'False'} : Time;
   //    IN : Bool := FALSE;
   //    Q { ExternalWritable := 'False'} : Bool;
   // END_VAR
BEGIN
END_DATA_BLOCK

DATA_BLOCK "CYL 10 DIR B TON"   // DB52
{ S7_Optimized_Access := 'TRUE' }
// stored: AutoNumber true, DBAccessibleFromOPCUA true, DBAccessibleFromWebserver true, InstanceOfName IEC_TIMER, OfSystemLibElement IEC_TIMER, OfSystemLibVersion 1.0
"IEC_TIMER"
   // VAR
   //    PT : Time := T#0MS;
   //    ET { ExternalWritable := 'False'} : Time;
   //    IN : Bool := FALSE;
   //    Q { ExternalWritable := 'False'} : Bool;
   // END_VAR
BEGIN
END_DATA_BLOCK

DATA_BLOCK "FC_EKS_R_TRIG_0"   // DB8200
// stored: AutoNumber true, DBAccessibleFromOPCUA true, DBAccessibleFromWebserver true, InstanceOfName R_TRIG, OfSystemLibElement R_TRIG, OfSystemLibVersion 1.0
"R_TRIG"
   // VAR_INPUT
   //    CLK : Bool := FALSE;
   // END_VAR
   // VAR_OUTPUT
   //    Q : Bool := FALSE;
   // END_VAR
   // VAR
   //    Stat_Bit : Bool := FALSE;
   // END_VAR
BEGIN
END_DATA_BLOCK

DATA_BLOCK "IEC_Timer_0_DB"   // DB13
{ S7_Optimized_Access := 'TRUE' }
// stored: AutoNumber true, DBAccessibleFromOPCUA true, DBAccessibleFromWebserver true, InstanceOfName IEC_TIMER, OfSystemLibElement IEC_TIMER, OfSystemLibVersion 1.0
"IEC_TIMER"
   // VAR
   //    PT : Time := T#2S;
   //    ET { ExternalWritable := 'False'} : Time;
   //    IN : Bool := FALSE;
   //    Q { ExternalWritable := 'False'} : Bool;
   // END_VAR
BEGIN
END_DATA_BLOCK

DATA_BLOCK "IEC_Timer_0_DB_1"   // DB64
{ S7_Optimized_Access := 'TRUE' }
// stored: AutoNumber true, DBAccessibleFromOPCUA true, DBAccessibleFromWebserver true, InstanceOfName IEC_TIMER, OfSystemLibElement IEC_TIMER, OfSystemLibVersion 1.0
"IEC_TIMER"
   // VAR
   //    PT : Time := T#2S;
   //    ET { ExternalWritable := 'False'} : Time;
   //    IN : Bool := FALSE;
   //    Q { ExternalWritable := 'False'} : Bool;
   // END_VAR
BEGIN
END_DATA_BLOCK

DATA_BLOCK "IEC_Timer_0_DB_10"   // DB18
{ S7_Optimized_Access := 'TRUE' }
// stored: AutoNumber true, DBAccessibleFromOPCUA true, DBAccessibleFromWebserver true, InstanceOfName IEC_TIMER, OfSystemLibElement IEC_TIMER, OfSystemLibVersion 1.0
"IEC_TIMER"
   // VAR
   //    PT : Time := T#5S;
   //    ET { ExternalWritable := 'False'} : Time;
   //    IN : Bool := TRUE;
   //    Q { ExternalWritable := 'False'} : Bool;
   // END_VAR
BEGIN
END_DATA_BLOCK

DATA_BLOCK "IEC_Timer_0_DB_11"   // DB19
{ S7_Optimized_Access := 'TRUE' }
// stored: AutoNumber true, DBAccessibleFromOPCUA true, DBAccessibleFromWebserver true, InstanceOfName IEC_TIMER, OfSystemLibElement IEC_TIMER, OfSystemLibVersion 1.0
"IEC_TIMER"
   // VAR
   //    PT : Time := T#5S;
   //    ET { ExternalWritable := 'False'} : Time;
   //    IN : Bool := TRUE;
   //    Q { ExternalWritable := 'False'} : Bool;
   // END_VAR
BEGIN
END_DATA_BLOCK

DATA_BLOCK "IEC_Timer_0_DB_12"   // DB22
{ S7_Optimized_Access := 'TRUE' }
// stored: AutoNumber true, DBAccessibleFromOPCUA true, DBAccessibleFromWebserver true, InstanceOfName IEC_TIMER, OfSystemLibElement IEC_TIMER, OfSystemLibVersion 1.0
"IEC_TIMER"
   // VAR
   //    PT : Time := T#0MS;
   //    ET { ExternalWritable := 'False'} : Time;
   //    IN : Bool := FALSE;
   //    Q { ExternalWritable := 'False'} : Bool;
   // END_VAR
BEGIN
END_DATA_BLOCK

DATA_BLOCK "IEC_Timer_0_DB_2"   // DB65
{ S7_Optimized_Access := 'TRUE' }
// stored: AutoNumber true, DBAccessibleFromOPCUA true, DBAccessibleFromWebserver true, InstanceOfName IEC_TIMER, OfSystemLibElement IEC_TIMER, OfSystemLibVersion 1.0
"IEC_TIMER"
   // VAR
   //    PT : Time := T#2S;
   //    ET { ExternalWritable := 'False'} : Time;
   //    IN : Bool := FALSE;
   //    Q { ExternalWritable := 'False'} : Bool;
   // END_VAR
BEGIN
END_DATA_BLOCK

DATA_BLOCK "IEC_Timer_0_DB_3"   // DB14
{ S7_Optimized_Access := 'TRUE' }
// stored: AutoNumber true, DBAccessibleFromOPCUA true, DBAccessibleFromWebserver true, InstanceOfName IEC_TIMER, OfSystemLibElement IEC_TIMER, OfSystemLibVersion 1.0
"IEC_TIMER"
   // VAR
   //    PT : Time := T#2S;
   //    ET { ExternalWritable := 'False'} : Time;
   //    IN : Bool := FALSE;
   //    Q { ExternalWritable := 'False'} : Bool;
   // END_VAR
BEGIN
END_DATA_BLOCK

DATA_BLOCK "IEC_Timer_0_DB_4"   // DB20
{ S7_Optimized_Access := 'TRUE' }
// stored: AutoNumber true, DBAccessibleFromOPCUA true, DBAccessibleFromWebserver true, InstanceOfName IEC_TIMER, OfSystemLibElement IEC_TIMER, OfSystemLibVersion 1.0
"IEC_TIMER"
   // VAR
   //    PT : Time := T#7S;
   //    ET { ExternalWritable := 'False'} : Time;
   //    IN : Bool := FALSE;
   //    Q { ExternalWritable := 'False'} : Bool;
   // END_VAR
BEGIN
END_DATA_BLOCK

DATA_BLOCK "IEC_Timer_0_DB_5"   // DB21
{ S7_Optimized_Access := 'TRUE' }
// stored: AutoNumber true, DBAccessibleFromOPCUA true, DBAccessibleFromWebserver true, InstanceOfName IEC_TIMER, OfSystemLibElement IEC_TIMER, OfSystemLibVersion 1.0
"IEC_TIMER"
   // VAR
   //    PT : Time := T#5S;
   //    ET { ExternalWritable := 'False'} : Time;
   //    IN : Bool := FALSE;
   //    Q { ExternalWritable := 'False'} : Bool;
   // END_VAR
BEGIN
END_DATA_BLOCK

DATA_BLOCK "IEC_Timer_0_DB_6"   // DB24
{ S7_Optimized_Access := 'TRUE' }
// stored: AutoNumber true, DBAccessibleFromOPCUA true, DBAccessibleFromWebserver true, InstanceOfName IEC_TIMER, OfSystemLibElement IEC_TIMER, OfSystemLibVersion 1.0
"IEC_TIMER"
   // VAR
   //    PT : Time := T#5S;
   //    ET { ExternalWritable := 'False'} : Time;
   //    IN : Bool := FALSE;
   //    Q { ExternalWritable := 'False'} : Bool;
   // END_VAR
BEGIN
END_DATA_BLOCK

DATA_BLOCK "IEC_Timer_0_DB_7"   // DB25
{ S7_Optimized_Access := 'TRUE' }
// stored: AutoNumber true, DBAccessibleFromOPCUA true, DBAccessibleFromWebserver true, InstanceOfName IEC_TIMER, OfSystemLibElement IEC_TIMER, OfSystemLibVersion 1.0
"IEC_TIMER"
   // VAR
   //    PT : Time := T#5S;
   //    ET { ExternalWritable := 'False'} : Time;
   //    IN : Bool := FALSE;
   //    Q { ExternalWritable := 'False'} : Bool;
   // END_VAR
BEGIN
END_DATA_BLOCK

DATA_BLOCK "IEC_Timer_0_DB_8"   // DB26
{ S7_Optimized_Access := 'TRUE' }
// stored: AutoNumber true, DBAccessibleFromOPCUA true, DBAccessibleFromWebserver true, InstanceOfName IEC_TIMER, OfSystemLibElement IEC_TIMER, OfSystemLibVersion 1.0
"IEC_TIMER"
   // VAR
   //    PT : Time := T#2S;
   //    ET { ExternalWritable := 'False'} : Time;
   //    IN : Bool := FALSE;
   //    Q { ExternalWritable := 'False'} : Bool;
   // END_VAR
BEGIN
END_DATA_BLOCK

DATA_BLOCK "IEC_Timer_0_DB_9"   // DB27
{ S7_Optimized_Access := 'TRUE' }
// stored: AutoNumber true, DBAccessibleFromOPCUA true, DBAccessibleFromWebserver true, InstanceOfName IEC_TIMER, OfSystemLibElement IEC_TIMER, OfSystemLibVersion 1.0
"IEC_TIMER"
   // VAR
   //    PT : Time := T#0MS;
   //    ET { ExternalWritable := 'False'} : Time;
   //    IN : Bool := FALSE;
   //    Q { ExternalWritable := 'False'} : Bool;
   // END_VAR
BEGIN
END_DATA_BLOCK

DATA_BLOCK "OPERATOR TEXT INDICATOR TIMER"   // DB9
{ S7_Optimized_Access := 'TRUE' }
// stored: AutoNumber true, DBAccessibleFromOPCUA true, DBAccessibleFromWebserver true, InstanceOfName IEC_TIMER, OfSystemLibElement IEC_TIMER, OfSystemLibVersion 1.0
"IEC_TIMER"
   // VAR
   //    PT : Time := T#800MS;
   //    ET { ExternalWritable := 'False'} : Time;
   //    IN : Bool := FALSE;
   //    Q { ExternalWritable := 'False'} : Bool;
   // END_VAR
BEGIN
END_DATA_BLOCK

DATA_BLOCK "PREASSURE_SENSOR_TIMER"   // DB16
{ S7_Optimized_Access := 'TRUE' }
// stored: AutoNumber true, DBAccessibleFromOPCUA true, DBAccessibleFromWebserver true, InstanceOfName IEC_TIMER, OfSystemLibElement IEC_TIMER, OfSystemLibVersion 1.0
"IEC_TIMER"
   // VAR
   //    PT : Time := T#3S;
   //    ET { ExternalWritable := 'False'} : Time;
   //    IN : Bool := FALSE;
   //    Q { ExternalWritable := 'False'} : Bool;
   // END_VAR
BEGIN
END_DATA_BLOCK

DATA_BLOCK "STEP CHANGE TIMER"   // DB11
{ S7_Optimized_Access := 'TRUE' }
// stored: AutoNumber true, DBAccessibleFromOPCUA true, DBAccessibleFromWebserver true, InstanceOfName IEC_TIMER, OfSystemLibElement IEC_TIMER, OfSystemLibVersion 1.0
"IEC_TIMER"
   // VAR
   //    PT : Time := T#500MS;
   //    ET { ExternalWritable := 'False'} : Time;
   //    IN : Bool := FALSE;
   //    Q { ExternalWritable := 'False'} : Bool;
   // END_VAR
BEGIN
END_DATA_BLOCK

DATA_BLOCK "TONR CICLE TIME TIMER"   // DB17
{ S7_Optimized_Access := 'TRUE' }
// stored: AutoNumber true, DBAccessibleFromOPCUA true, DBAccessibleFromWebserver true, InstanceOfName IEC_TIMER, OfSystemLibElement IEC_TIMER, OfSystemLibVersion 1.0
"IEC_TIMER"
   // VAR
   //    PT : Time := T#2H;
   //    ET { ExternalWritable := 'False'} : Time;
   //    IN : Bool := FALSE;
   //    Q { ExternalWritable := 'False'} : Bool;
   // END_VAR
BEGIN
END_DATA_BLOCK

DATA_BLOCK "leftInsertionAlarmTimer"   // DB23
{ S7_Optimized_Access := 'TRUE' }
// stored: AutoNumber true, DBAccessibleFromOPCUA true, DBAccessibleFromWebserver true, InstanceOfName IEC_TIMER, OfSystemLibElement IEC_TIMER, OfSystemLibVersion 1.0
"IEC_TIMER"
   // VAR
   //    PT : Time := T#2S;
   //    ET { ExternalWritable := 'False'} : Time;
   //    IN : Bool := FALSE;
   //    Q { ExternalWritable := 'False'} : Bool;
   // END_VAR
BEGIN
END_DATA_BLOCK

DATA_BLOCK "rightInsertionAlarmTimer"   // DB28
{ S7_Optimized_Access := 'TRUE' }
// stored: AutoNumber true, DBAccessibleFromOPCUA true, DBAccessibleFromWebserver true, InstanceOfName IEC_TIMER, OfSystemLibElement IEC_TIMER, OfSystemLibVersion 1.0
"IEC_TIMER"
   // VAR
   //    PT : Time := T#5S;
   //    ET { ExternalWritable := 'False'} : Time;
   //    IN : Bool := FALSE;
   //    Q { ExternalWritable := 'False'} : Bool;
   // END_VAR
BEGIN
END_DATA_BLOCK

DATA_BLOCK "trigger"   // DB33
{ S7_Optimized_Access := 'TRUE' }
// stored: AutoNumber true, DBAccessibleFromOPCUA true, DBAccessibleFromWebserver true, InstanceOfName IEC_TIMER, OfSystemLibElement IEC_TIMER, OfSystemLibVersion 1.0
"IEC_TIMER"
   // VAR
   //    PT : Time := T#20MS;
   //    ET { ExternalWritable := 'False'} : Time;
   //    IN : Bool := TRUE;
   //    Q { ExternalWritable := 'False'} : Bool;
   // END_VAR
BEGIN
END_DATA_BLOCK

DATA_BLOCK "DB_INST_AWAKE_SIGNAL"   // DB1003
VERSION : 0.1
// stored: AutoNumber false, DBAccessibleFromOPCUA true, DBAccessibleFromWebserver true, InstanceOfName FB_IJC_AWAKE_SIGNAL, InstanceOfType FB
"FB_IJC_AWAKE_SIGNAL"
BEGIN
END_DATA_BLOCK

